LIN {X 0,Y 516.191,Z 499.318,A -85,B 0,C 180,E1 -4981.156,E2 -4981.156} C_VEL
LIN {X 0,Y 516.198,Z 499.528,A -85,B 0,C 180,E1 -4982.421,E2 -4982.421} C_VEL
LIN {X 0,Y 516.212,Z 498.459,A -85,B 0,C 180,E1 -4983.931,E2 -4983.931} C_VEL
LIN {X 0,Y 516.231,Z 496.319,A -85,B 0,C 180,E1 -4985.229,E2 -4985.229} C_VEL
LIN {X 0,Y 516.336,Z 492.856,A -85,B 0,C 180,E1 -4986.576,E2 -4986.576} C_VEL
LIN {X 0,Y 516.422,Z 488.222,A -85,B 0,C 180,E1 -4987.877,E2 -4987.877} C_VEL
LIN {X 0,Y 516.57,Z 482.317,A -85,B 0,C 180,E1 -4989.15,E2 -4989.15} C_VEL
LIN {X 0,Y 516.77,Z 474.967,A -85,B 0,C 180,E1 -4990.395,E2 -4990.395} C_VEL
LIN {X 0,Y 516.949,Z 467.344,A -85,B 0,C 180,E1 -4991.437,E2 -4991.437} C_VEL
LIN {X 0,Y 517.264,Z 457.539,A -85,B 0,C 180,E1 -4992.527,E2 -4992.527} C_VEL
LIN {X 0,Y 517.546,Z 447.499,A -85,B 0,C 180,E1 -4993.428,E2 -4993.428} C_VEL
LIN {X 0,Y 517.803,Z 437.525,A -85,B 0,C 180,E1 -4994.151,E2 -4994.151} C_VEL
LIN {X 0,Y 518.099,Z 426.299,A -85,B 0,C 180,E1 -4994.797,E2 -4994.797} C_VEL
LIN {X 0,Y 518.372,Z 414.041,A -85,B 0,C 180,E1 -4995.333,E2 -4995.333} C_VEL
LIN {X 0,Y 518.246,Z 407.392,A -85,B 0,C 180,E1 -4995.565,E2 -4995.565} C_VEL
LIN {X 0,Y 516.248,Z 397.17,A -85,B 0,C 180,E1 -4995.893,E2 -4995.893} C_VEL
LIN {X 0,Y 516.275,Z 394.338,A -85,B 0,C 180,E1 -4998.478,E2 -4998.478} C_VEL
LIN {X 0,Y 516.29,Z 391.343,A -85,B 0,C 180,E1 -5001.231,E2 -5001.231} C_VEL
LIN {X 0,Y 516.378,Z 388.125,A -85,B 0,C 180,E1 -5004.18,E2 -5004.18} C_VEL
LIN {X 0,Y 516.457,Z 385.062,A -85,B 0,C 180,E1 -5007.021,E2 -5007.021} C_VEL
LIN {X 0,Y 516.53,Z 382.092,A -85,B 0,C 180,E1 -5009.773,E2 -5009.773} C_VEL
LIN {X 0,Y 516.548,Z 379.223,A -85,B 0,C 180,E1 -5012.445,E2 -5012.445} C_VEL
LIN {X 0,Y 516.602,Z 376.37,A -85,B 0,C 180,E1 -5015.056,E2 -5015.056} C_VEL
LIN {X 0,Y 516.777,Z 376.119,A -85,B 0,C 180,E1 -5016.772,E2 -5016.772} C_VEL
LIN {X 0,Y 516.934,Z 376.098,A -85,B 0,C 180,E1 -5019.731,E2 -5019.731} C_VEL
LIN {X 0,Y 516.923,Z 376.096,A -85,B 0,C 180,E1 -5022.596,E2 -5022.596} C_VEL
LIN {X 0,Y 516.936,Z 376.095,A -85,B 0,C 180,E1 -5025.03,E2 -5025.03} C_VEL
LIN {X 0,Y 516.959,Z 376.094,A -85,B 0,C 180,E1 -5028.233,E2 -5028.233} C_VEL
LIN {X 0,Y 516.964,Z 376.091,A -85,B 0,C 180,E1 -5031.399,E2 -5031.399} C_VEL
LIN {X 0,Y 517.004,Z 376.086,A -85,B 0,C 180,E1 -5033.757,E2 -5033.757} C_VEL
LIN {X 0,Y 517.079,Z 376.076,A -85,B 0,C 180,E1 -5037.663,E2 -5037.663} C_VEL
LIN {X 0,Y 517.09,Z 376.075,A -85,B 0,C 180,E1 -5040.779,E2 -5040.779} C_VEL
LIN {X 0,Y 517.009,Z 376.086,A -85,B 0,C 180,E1 -5043.117,E2 -5043.117} C_VEL
LIN {X 0,Y 517.003,Z 376.087,A -85,B 0,C 180,E1 -5046.243,E2 -5046.243} C_VEL
LIN {X 0,Y 516.949,Z 376.092,A -85,B 0,C 180,E1 -5049.389,E2 -5049.389} C_VEL
LIN {X 0,Y 516.951,Z 376.092,A -85,B 0,C 180,E1 -5051.81,E2 -5051.81} C_VEL
LIN {X 0,Y 516.938,Z 376.094,A -85,B 0,C 180,E1 -5055.147,E2 -5055.147} C_VEL
LIN {X 0,Y 516.92,Z 376.097,A -85,B 0,C 180,E1 -5058.222,E2 -5058.222} C_VEL
LIN {X 0,Y 516.906,Z 376.099,A -85,B 0,C 180,E1 -5060.702,E2 -5060.702} C_VEL
LIN {X 0,Y 516.906,Z 376.098,A -85,B 0,C 180,E1 -5064.072,E2 -5064.072} C_VEL
LIN {X 0,Y 516.924,Z 376.095,A -85,B 0,C 180,E1 -5066.658,E2 -5066.658} C_VEL
LIN {X 0,Y 516.906,Z 376.101,A -85,B 0,C 180,E1 -5069.524,E2 -5069.524} C_VEL
LIN {X 0,Y 516.889,Z 376.101,A -85,B 0,C 180,E1 -5072.543,E2 -5072.543} C_VEL
LIN {X 0,Y 516.862,Z 376.106,A -85,B 0,C 180,E1 -5075.33,E2 -5075.33} C_VEL
LIN {X 0,Y 516.877,Z 376.105,A -85,B 0,C 180,E1 -5077.944,E2 -5077.944} C_VEL
LIN {X 0,Y 516.901,Z 376.1,A -85,B 0,C 180,E1 -5080.74,E2 -5080.74} C_VEL
LIN {X 0,Y 516.879,Z 376.105,A -85,B 0,C 180,E1 -5083.904,E2 -5083.904} C_VEL
LIN {X 0,Y 516.88,Z 376.104,A -85,B 0,C 180,E1 -5086.107,E2 -5086.107} C_VEL
LIN {X 0,Y 516.894,Z 376.102,A -85,B 0,C 180,E1 -5089.26,E2 -5089.26} C_VEL
LIN {X 0,Y 516.898,Z 376.203,A -85,B 0,C 180,E1 -5091.227,E2 -5091.227} C_VEL
LIN {X 0,Y 518.101,Z 382.793,A -85,B 0,C 180,E1 -5093.838,E2 -5093.838} C_VEL
LIN {X 0,Y 518.058,Z 388.209,A -85,B 0,C 180,E1 -5095.846,E2 -5095.846} C_VEL
LIN {X 0,Y 517.781,Z 396.952,A -85,B 0,C 180,E1 -5098.773,E2 -5098.773} C_VEL
LIN {X 0,Y 517.567,Z 406.705,A -85,B 0,C 180,E1 -5101.962,E2 -5101.962} C_VEL
LIN {X 0,Y 517.319,Z 414.959,A -85,B 0,C 180,E1 -5104.663,E2 -5104.663} C_VEL
LIN {X 0,Y 517.116,Z 424.226,A -85,B 0,C 180,E1 -5107.633,E2 -5107.633} C_VEL
LIN {X 0,Y 516.907,Z 433.493,A -85,B 0,C 180,E1 -5110.543,E2 -5110.543} C_VEL
LIN {X 0,Y 516.712,Z 442.76,A -85,B 0,C 180,E1 -5113.404,E2 -5113.404} C_VEL
LIN {X 0,Y 516.591,Z 451.736,A -85,B 0,C 180,E1 -5116.095,E2 -5116.095} C_VEL
LIN {X 0,Y 518.517,Z 464.185,A -85,B 0,C 180,E1 -5116.429,E2 -5116.429} C_VEL
LIN {X 0,Y 518.247,Z 476.985,A -85,B 0,C 180,E1 -5116.871,E2 -5116.871} C_VEL
LIN {X 0,Y 517.949,Z 489.176,A -85,B 0,C 180,E1 -5117.461,E2 -5117.461} C_VEL
LIN {X 0,Y 517.703,Z 500.576,A -85,B 0,C 180,E1 -5118.179,E2 -5118.179} C_VEL
LIN {X 0,Y 517.38,Z 511.401,A -85,B 0,C 180,E1 -5119.037,E2 -5119.037} C_VEL
LIN {X 0,Y 517.045,Z 521.335,A -85,B 0,C 180,E1 -5120.02,E2 -5120.02} C_VEL
LIN {X 0,Y 516.814,Z 530.96,A -85,B 0,C 180,E1 -5121.2,E2 -5121.2} C_VEL
LIN {X 0,Y 516.563,Z 538.621,A -85,B 0,C 180,E1 -5122.377,E2 -5122.377} C_VEL
LIN {X 0,Y 516.427,Z 545.679,A -85,B 0,C 180,E1 -5123.75,E2 -5123.75} C_VEL
LIN {X 0,Y 516.313,Z 550.372,A -85,B 0,C 180,E1 -5124.924,E2 -5124.924} C_VEL
LIN {X 0,Y 516.355,Z 553.957,A -85,B 0,C 180,E1 -5126.098,E2 -5126.098} C_VEL
LIN {X 0,Y 516.282,Z 555.807,A -85,B 0,C 180,E1 -5126.879,E2 -5126.879} C_VEL
LIN {X 0,Y 516.261,Z 557.196,A -85,B 0,C 180,E1 -5127.659,E2 -5127.659} C_VEL
LIN {X 0,Y 516.16,Z 558.785,A -85,B 0,C 180,E1 -5129.22,E2 -5129.22} C_VEL
LIN {X 0,Y 516.154,Z 559,A -85,B 0,C 180,E1 -5130,E2 -5130} C_VEL
LIN {X 0,Y 516.192,Z 558.186,A -85,B 0,C 180,E1 -5131.56,E2 -5131.56} C_VEL
LIN {X 0,Y 516.261,Z 557.199,A -85,B 0,C 180,E1 -5132.34,E2 -5132.34} C_VEL
LIN {X 0,Y 516.282,Z 555.81,A -85,B 0,C 180,E1 -5133.121,E2 -5133.121} C_VEL
LIN {X 0,Y 516.344,Z 552.896,A -85,B 0,C 180,E1 -5134.293,E2 -5134.293} C_VEL
LIN {X 0,Y 516.405,Z 548.95,A -85,B 0,C 180,E1 -5135.466,E2 -5135.466} C_VEL
LIN {X 0,Y 516.486,Z 543.035,A -85,B 0,C 180,E1 -5136.807,E2 -5136.807} C_VEL
LIN {X 0,Y 516.64,Z 536.239,A -85,B 0,C 180,E1 -5138.015,E2 -5138.015} C_VEL
LIN {X 0,Y 516.867,Z 527.994,A -85,B 0,C 180,E1 -5139.193,E2 -5139.193} C_VEL
LIN {X 0,Y 517.078,Z 519.543,A -85,B 0,C 180,E1 -5140.177,E2 -5140.177} C_VEL
LIN {X 0,Y 517.474,Z 509.101,A -85,B 0,C 180,E1 -5141.159,E2 -5141.159} C_VEL
LIN {X 0,Y 517.718,Z 497.634,A -85,B 0,C 180,E1 -5142.026,E2 -5142.026} C_VEL
LIN {X 0,Y 517.981,Z 487.416,A -85,B 0,C 180,E1 -5142.637,E2 -5142.637} C_VEL
LIN {X 0,Y 518.269,Z 475.776,A -85,B 0,C 180,E1 -5143.178,E2 -5143.178} C_VEL
LIN {X 0,Y 518.44,Z 462.821,A -85,B 0,C 180,E1 -5143.61,E2 -5143.61} C_VEL
LIN {X 0,Y 516.574,Z 451.532,A -85,B 0,C 180,E1 -5143.924,E2 -5143.924} C_VEL
LIN {X 0,Y 516.712,Z 442.761,A -85,B 0,C 180,E1 -5146.596,E2 -5146.596} C_VEL
LIN {X 0,Y 516.906,Z 433.494,A -85,B 0,C 180,E1 -5149.457,E2 -5149.457} C_VEL
LIN {X 0,Y 517.096,Z 423.966,A -85,B 0,C 180,E1 -5152.45,E2 -5152.45} C_VEL
LIN {X 0,Y 517.371,Z 413.636,A -85,B 0,C 180,E1 -5155.765,E2 -5155.765} C_VEL
LIN {X 0,Y 517.598,Z 404.312,A -85,B 0,C 180,E1 -5158.817,E2 -5158.817} C_VEL
LIN {X 0,Y 517.836,Z 396.125,A -85,B 0,C 180,E1 -5161.547,E2 -5161.547} C_VEL
LIN {X 0,Y 518.098,Z 388.482,A -85,B 0,C 180,E1 -5164.161,E2 -5164.161} C_VEL
LIN {X 0,Y 518.11,Z 382.817,A -85,B 0,C 180,E1 -5166.16,E2 -5166.16} C_VEL
LIN {X 0,Y 516.893,Z 376.1,A -85,B 0,C 180,E1 -5168.892,E2 -5168.892} C_VEL
LIN {X 0,Y 516.91,Z 376.099,A -85,B 0,C 180,E1 -5171.774,E2 -5171.774} C_VEL
LIN {X 0,Y 516.918,Z 376.099,A -85,B 0,C 180,E1 -5175.009,E2 -5175.009} C_VEL
LIN {X 0,Y 516.917,Z 376.099,A -85,B 0,C 180,E1 -5178.397,E2 -5178.397} C_VEL
LIN {X 0,Y 516.881,Z 376.102,A -85,B 0,C 180,E1 -5181.284,E2 -5181.284} C_VEL
LIN {X 0,Y 516.885,Z 376.102,A -85,B 0,C 180,E1 -5184.221,E2 -5184.221} C_VEL
LIN {X 0,Y 516.892,Z 376.102,A -85,B 0,C 180,E1 -5187.053,E2 -5187.053} C_VEL
LIN {X 0,Y 516.885,Z 376.1,A -85,B 0,C 180,E1 -5189.796,E2 -5189.796} C_VEL
LIN {X 0,Y 516.923,Z 376.096,A -85,B 0,C 180,E1 -5192.467,E2 -5192.467} C_VEL
LIN {X 0,Y 516.903,Z 376.101,A -85,B 0,C 180,E1 -5195.071,E2 -5195.071} C_VEL
LIN {X 0,Y 516.878,Z 376.104,A -85,B 0,C 180,E1 -5198.462,E2 -5198.462} C_VEL
LIN {X 0,Y 516.897,Z 376.1,A -85,B 0,C 180,E1 -5200.955,E2 -5200.955} C_VEL
LIN {X 0,Y 516.909,Z 376.098,A -85,B 0,C 180,E1 -5203.41,E2 -5203.41} C_VEL
LIN {X 0,Y 516.886,Z 376.101,A -85,B 0,C 180,E1 -5205.833,E2 -5205.833} C_VEL
LIN {X 0,Y 516.948,Z 376.094,A -85,B 0,C 180,E1 -5209.028,E2 -5209.028} C_VEL
LIN {X 0,Y 516.97,Z 376.09,A -85,B 0,C 180,E1 -5212.187,E2 -5212.187} C_VEL
LIN {X 0,Y 517.02,Z 376.085,A -85,B 0,C 180,E1 -5214.54,E2 -5214.54} C_VEL
LIN {X 0,Y 517.074,Z 376.076,A -85,B 0,C 180,E1 -5217.663,E2 -5217.663} C_VEL
LIN {X 0,Y 517.088,Z 376.076,A -85,B 0,C 180,E1 -5220.779,E2 -5220.779} C_VEL
LIN {X 0,Y 517.008,Z 376.085,A -85,B 0,C 180,E1 -5223.117,E2 -5223.117} C_VEL
LIN {X 0,Y 517.002,Z 376.088,A -85,B 0,C 180,E1 -5226.243,E2 -5226.243} C_VEL
LIN {X 0,Y 516.95,Z 376.093,A -85,B 0,C 180,E1 -5229.389,E2 -5229.389} C_VEL
LIN {X 0,Y 516.948,Z 376.094,A -85,B 0,C 180,E1 -5231.811,E2 -5231.811} C_VEL
LIN {X 0,Y 516.935,Z 376.094,A -85,B 0,C 180,E1 -5235.147,E2 -5235.147} C_VEL
LIN {X 0,Y 516.917,Z 376.099,A -85,B 0,C 180,E1 -5238.223,E2 -5238.223} C_VEL
LIN {X 0,Y 516.905,Z 376.099,A -85,B 0,C 180,E1 -5240.702,E2 -5240.702} C_VEL
LIN {X 0,Y 516.903,Z 376.1,A -85,B 0,C 180,E1 -5244.073,E2 -5244.073} C_VEL
LIN {X 0,Y 516.922,Z 376.097,A -85,B 0,C 180,E1 -5246.658,E2 -5246.658} C_VEL
LIN {X 0,Y 516.904,Z 376.099,A -85,B 0,C 180,E1 -5249.525,E2 -5249.525} C_VEL
LIN {X 0,Y 516.895,Z 376.102,A -85,B 0,C 180,E1 -5252.545,E2 -5252.545} C_VEL
LIN {X 0,Y 516.879,Z 376.1,A -85,B 0,C 180,E1 -5255.333,E2 -5255.333} C_VEL
LIN {X 0,Y 516.877,Z 376.103,A -85,B 0,C 180,E1 -5257.944,E2 -5257.944} C_VEL
LIN {X 0,Y 516.9,Z 376.099,A -85,B 0,C 180,E1 -5260.74,E2 -5260.74} C_VEL
LIN {X 0,Y 516.878,Z 376.103,A -85,B 0,C 180,E1 -5263.904,E2 -5263.904} C_VEL
LIN {X 0,Y 516.879,Z 376.103,A -85,B 0,C 180,E1 -5266.108,E2 -5266.108} C_VEL
LIN {X 0,Y 516.915,Z 376.098,A -85,B 0,C 180,E1 -5268.399,E2 -5268.399} C_VEL
LIN {X 0,Y 516.879,Z 376.104,A -85,B 0,C 180,E1 -5270.307,E2 -5270.307} C_VEL
LIN {X 0,Y 516.21,Z 376.185,A -85,B 0,C 180,E1 -5270.957,E2 -5270.957} C_VEL
LIN {X 0,Y 513.365,Z 376.54,A -85,B 0,C 180,E1 -5272.013,E2 -5272.013} C_VEL
LIN {X 0,Y 510.957,Z 376.842,A -85,B 0,C 180,E1 -5272.863,E2 -5272.863} C_VEL
LIN {X 0,Y 509.917,Z 376.971,A -85,B 0,C 180,E1 -5273.52,E2 -5273.52} C_VEL
LIN {X 0,Y 509.828,Z 376.981,A -85,B 0,C 180,E1 -5273.742,E2 -5273.742} C_VEL
LIN {X 0,Y 509.861,Z 376.977,A -85,B 0,C 180,E1 -5276.54,E2 -5276.54} C_VEL
LIN {X 0,Y 509.846,Z 376.979,A -85,B 0,C 180,E1 -5279.335,E2 -5279.335} C_VEL
LIN {X 0,Y 509.894,Z 376.973,A -85,B 0,C 180,E1 -5282.055,E2 -5282.055} C_VEL
LIN {X 0,Y 509.879,Z 376.974,A -85,B 0,C 180,E1 -5284.705,E2 -5284.705} C_VEL
LIN {X 0,Y 509.839,Z 376.979,A -85,B 0,C 180,E1 -5287.456,E2 -5287.456} C_VEL
LIN {X 0,Y 509.919,Z 376.969,A -85,B 0,C 180,E1 -5289.845,E2 -5289.845} C_VEL
LIN {X 0,Y 509.883,Z 376.972,A -85,B 0,C 180,E1 -5293.175,E2 -5293.175} C_VEL
LIN {X 0,Y 509.868,Z 376.976,A -85,B 0,C 180,E1 -5295.635,E2 -5295.635} C_VEL
LIN {X 0,Y 509.917,Z 376.969,A -85,B 0,C 180,E1 -5298.875,E2 -5298.875} C_VEL
LIN {X 0,Y 509.955,Z 376.965,A -85,B 0,C 180,E1 -5302.079,E2 -5302.079} C_VEL
LIN {X 0,Y 509.986,Z 376.961,A -85,B 0,C 180,E1 -5304.465,E2 -5304.465} C_VEL
LIN {X 0,Y 509.828,Z 376.984,A -85,B 0,C 180,E1 -5308.42,E2 -5308.42} C_VEL
LIN {X 0,Y 509.779,Z 376.991,A -85,B 0,C 180,E1 -5309.21,E2 -5309.21} C_VEL
LIN {X 0,Y 509.632,Z 378.352,A -85,B 0,C 180,E1 -5310.79,E2 -5310.79} C_VEL
LIN {X 0,Y 509.491,Z 382.661,A -85,B 0,C 180,E1 -5314.748,E2 -5314.748} C_VEL
LIN {X 0,Y 509.445,Z 385.291,A -85,B 0,C 180,E1 -5317.132,E2 -5317.132} C_VEL
LIN {X 0,Y 509.358,Z 388.826,A -85,B 0,C 180,E1 -5320.333,E2 -5320.333} C_VEL
LIN {X 0,Y 509.291,Z 391.515,A -85,B 0,C 180,E1 -5322.756,E2 -5322.756} C_VEL
LIN {X 0,Y 509.302,Z 394.318,A -85,B 0,C 180,E1 -5325.2,E2 -5325.2} C_VEL
LIN {X 0,Y 509.21,Z 397.43,A -85,B 0,C 180,E1 -5328.014,E2 -5328.014} C_VEL
LIN {X 0,Y 511.466,Z 408.493,A -85,B 0,C 180,E1 -5328.372,E2 -5328.372} C_VEL
LIN {X 0,Y 511.353,Z 420.799,A -85,B 0,C 180,E1 -5328.843,E2 -5328.843} C_VEL
LIN {X 0,Y 511.021,Z 433.18,A -85,B 0,C 180,E1 -5329.482,E2 -5329.482} C_VEL
LIN {X 0,Y 510.748,Z 444.58,A -85,B 0,C 180,E1 -5330.256,E2 -5330.256} C_VEL
LIN {X 0,Y 510.386,Z 455.513,A -85,B 0,C 180,E1 -5331.19,E2 -5331.19} C_VEL
LIN {X 0,Y 510.048,Z 465.493,A -85,B 0,C 180,E1 -5332.253,E2 -5332.253} C_VEL
LIN {X 0,Y 509.729,Z 473.801,A -85,B 0,C 180,E1 -5333.353,E2 -5333.353} C_VEL
LIN {X 0,Y 509.56,Z 481.606,A -85,B 0,C 180,E1 -5334.637,E2 -5334.637} C_VEL
LIN {X 0,Y 509.419,Z 487.051,A -85,B 0,C 180,E1 -5335.758,E2 -5335.758} C_VEL
LIN {X 0,Y 509.286,Z 492.135,A -85,B 0,C 180,E1 -5337.09,E2 -5337.09} C_VEL
LIN {X 0,Y 509.216,Z 495.877,A -85,B 0,C 180,E1 -5338.434,E2 -5338.434} C_VEL
LIN {X 0,Y 509.151,Z 498.412,A -85,B 0,C 180,E1 -5339.796,E2 -5339.796} C_VEL
LIN {X 0,Y 509.114,Z 499.749,A -85,B 0,C 180,E1 -5341.143,E2 -5341.143} C_VEL
LIN {X 0,Y 509.103,Z 499.922,A -85,B 0,C 180,E1 -5342.639,E2 -5342.639} C_VEL
LIN {X 0,Y 509.122,Z 498.729,A -85,B 0,C 180,E1 -5344.08,E2 -5344.08} C_VEL
LIN {X 0,Y 509.184,Z 496.303,A -85,B 0,C 180,E1 -5345.477,E2 -5345.477} C_VEL
LIN {X 0,Y 509.281,Z 492.696,A -85,B 0,C 180,E1 -5346.832,E2 -5346.832} C_VEL
LIN {X 0,Y 509.403,Z 487.894,A -85,B 0,C 180,E1 -5348.149,E2 -5348.149} C_VEL
LIN {X 0,Y 509.573,Z 481.777,A -85,B 0,C 180,E1 -5349.434,E2 -5349.434} C_VEL
LIN {X 0,Y 509.787,Z 474.19,A -85,B 0,C 180,E1 -5350.69,E2 -5350.69} C_VEL
LIN {X 0,Y 510.061,Z 465.702,A -85,B 0,C 180,E1 -5351.823,E2 -5351.823} C_VEL
LIN {X 0,Y 510.323,Z 456.477,A -85,B 0,C 180,E1 -5352.822,E2 -5352.822} C_VEL
LIN {X 0,Y 510.672,Z 445.775,A -85,B 0,C 180,E1 -5353.752,E2 -5353.752} C_VEL
LIN {X 0,Y 510.944,Z 434.354,A -85,B 0,C 180,E1 -5354.547,E2 -5354.547} C_VEL
LIN {X 0,Y 511.274,Z 422.583,A -85,B 0,C 180,E1 -5355.176,E2 -5355.176} C_VEL
LIN {X 0,Y 511.513,Z 409.334,A -85,B 0,C 180,E1 -5355.695,E2 -5355.695} C_VEL
LIN {X 0,Y 509.588,Z 399.448,A -85,B 0,C 180,E1 -5356.024,E2 -5356.024} C_VEL
LIN {X 0,Y 509.179,Z 397.637,A -85,B 0,C 180,E1 -5356.088,E2 -5356.088} C_VEL
LIN {X 0,Y 509.207,Z 394.981,A -85,B 0,C 180,E1 -5358.51,E2 -5358.51} C_VEL
LIN {X 0,Y 509.232,Z 391.61,A -85,B 0,C 180,E1 -5361.607,E2 -5361.607} C_VEL
LIN {X 0,Y 509.344,Z 388.36,A -85,B 0,C 180,E1 -5364.583,E2 -5364.583} C_VEL
LIN {X 0,Y 509.419,Z 385.318,A -85,B 0,C 180,E1 -5367.449,E2 -5367.449} C_VEL
LIN {X 0,Y 509.465,Z 382.195,A -85,B 0,C 180,E1 -5370.35,E2 -5370.35} C_VEL
LIN {X 0,Y 509.494,Z 379.428,A -85,B 0,C 180,E1 -5372.922,E2 -5372.922} C_VEL
LIN {X 0,Y 509.528,Z 377.548,A -85,B 0,C 180,E1 -5374.685,E2 -5374.685} C_VEL
LIN {X 0,Y 509.61,Z 377.01,A -85,B 0,C 180,E1 -5375.561,E2 -5375.561} C_VEL
LIN {X 0,Y 509.816,Z 376.984,A -85,B 0,C 180,E1 -5378.148,E2 -5378.148} C_VEL
LIN {X 0,Y 509.86,Z 376.978,A -85,B 0,C 180,E1 -5380.681,E2 -5380.681} C_VEL
LIN {X 0,Y 509.879,Z 376.975,A -85,B 0,C 180,E1 -5383.174,E2 -5383.174} C_VEL
LIN {X 0,Y 509.857,Z 376.978,A -85,B 0,C 180,E1 -5385.634,E2 -5385.634} C_VEL
LIN {X 0,Y 509.911,Z 376.969,A -85,B 0,C 180,E1 -5388.874,E2 -5388.874} C_VEL
LIN {X 0,Y 509.945,Z 376.965,A -85,B 0,C 180,E1 -5392.078,E2 -5392.078} C_VEL
LIN {X 0,Y 509.977,Z 376.961,A -85,B 0,C 180,E1 -5394.464,E2 -5394.464} C_VEL
LIN {X 0,Y 510.049,Z 376.952,A -85,B 0,C 180,E1 -5397.631,E2 -5397.631} C_VEL
LIN {X 0,Y 510.06,Z 376.951,A -85,B 0,C 180,E1 -5400.789,E2 -5400.789} C_VEL
LIN {X 0,Y 509.951,Z 376.964,A -85,B 0,C 180,E1 -5403.16,E2 -5403.16} C_VEL
LIN {X 0,Y 509.971,Z 376.964,A -85,B 0,C 180,E1 -5406.33,E2 -5406.33} C_VEL
LIN {X 0,Y 509.91,Z 376.971,A -85,B 0,C 180,E1 -5408.72,E2 -5408.72} C_VEL
LIN {X 0,Y 509.899,Z 376.971,A -85,B 0,C 180,E1 -5411.932,E2 -5411.932} C_VEL
LIN {X 0,Y 509.887,Z 376.972,A -85,B 0,C 180,E1 -5415.242,E2 -5415.242} C_VEL
LIN {X 0,Y 509.883,Z 376.972,A -85,B 0,C 180,E1 -5418.001,E2 -5418.001} C_VEL
LIN {X 0,Y 509.844,Z 376.98,A -85,B 0,C 180,E1 -5421.002,E2 -5421.002} C_VEL
LIN {X 0,Y 509.865,Z 376.977,A -85,B 0,C 180,E1 -5424.426,E2 -5424.426} C_VEL
LIN {X 0,Y 509.883,Z 376.975,A -85,B 0,C 180,E1 -5427.056,E2 -5427.056} C_VEL
LIN {X 0,Y 509.852,Z 376.978,A -85,B 0,C 180,E1 -5429.751,E2 -5429.751} C_VEL
LIN {X 0,Y 509.862,Z 376.978,A -85,B 0,C 180,E1 -5432.773,E2 -5432.773} C_VEL
LIN {X 0,Y 509.821,Z 376.985,A -85,B 0,C 180,E1 -5435.579,E2 -5435.579} C_VEL
LIN {X 0,Y 509.855,Z 376.977,A -85,B 0,C 180,E1 -5438.338,E2 -5438.338} C_VEL
LIN {X 0,Y 509.863,Z 376.978,A -85,B 0,C 180,E1 -5441.425,E2 -5441.425} C_VEL
LIN {X 0,Y 509.854,Z 376.977,A -85,B 0,C 180,E1 -5444.668,E2 -5444.668} C_VEL
LIN {X 0,Y 509.857,Z 376.979,A -85,B 0,C 180,E1 -5448.103,E2 -5448.103} C_VEL
LIN {X 0,Y 509.882,Z 377.132,A -85,B 0,C 180,E1 -5450.97,E2 -5450.97} C_VEL
LIN {X 0,Y 511.155,Z 384.063,A -85,B 0,C 180,E1 -5453.757,E2 -5453.757} C_VEL
LIN {X 0,Y 511.097,Z 389.175,A -85,B 0,C 180,E1 -5455.683,E2 -5455.683} C_VEL
LIN {X 0,Y 510.803,Z 397.429,A -85,B 0,C 180,E1 -5458.544,E2 -5458.544} C_VEL
LIN {X 0,Y 510.548,Z 407.134,A -85,B 0,C 180,E1 -5461.763,E2 -5461.763} C_VEL
LIN {X 0,Y 510.298,Z 416.282,A -85,B 0,C 180,E1 -5464.727,E2 -5464.727} C_VEL
LIN {X 0,Y 510.079,Z 425.674,A -85,B 0,C 180,E1 -5467.775,E2 -5467.775} C_VEL
LIN {X 0,Y 509.86,Z 434.817,A -85,B 0,C 180,E1 -5470.682,E2 -5470.682} C_VEL
LIN {X 0,Y 509.648,Z 445.408,A -85,B 0,C 180,E1 -5473.991,E2 -5473.991} C_VEL
LIN {X 0,Y 509.544,Z 451.736,A -85,B 0,C 180,E1 -5475.899,E2 -5475.899} C_VEL
LIN {X 0,Y 511.549,Z 464.185,A -85,B 0,C 180,E1 -5476.24,E2 -5476.24} C_VEL
LIN {X 0,Y 511.336,Z 476.985,A -85,B 0,C 180,E1 -5476.69,E2 -5476.69} C_VEL
LIN {X 0,Y 511.001,Z 489.175,A -85,B 0,C 180,E1 -5477.288,E2 -5477.288} C_VEL
LIN {X 0,Y 510.727,Z 499.95,A -85,B 0,C 180,E1 -5477.971,E2 -5477.971} C_VEL
LIN {X 0,Y 510.404,Z 511.4,A -85,B 0,C 180,E1 -5478.885,E2 -5478.885} C_VEL
LIN {X 0,Y 510.03,Z 521.334,A -85,B 0,C 180,E1 -5479.881,E2 -5479.881} C_VEL
LIN {X 0,Y 509.76,Z 530.96,A -85,B 0,C 180,E1 -5481.077,E2 -5481.077} C_VEL
LIN {X 0,Y 509.522,Z 538.621,A -85,B 0,C 180,E1 -5482.271,E2 -5482.271} C_VEL
LIN {X 0,Y 509.336,Z 545.679,A -85,B 0,C 180,E1 -5483.662,E2 -5483.662} C_VEL
LIN {X 0,Y 509.248,Z 550.372,A -85,B 0,C 180,E1 -5484.853,E2 -5484.853} C_VEL
LIN {X 0,Y 509.253,Z 553.958,A -85,B 0,C 180,E1 -5486.043,E2 -5486.043} C_VEL
LIN {X 0,Y 509.2,Z 555.807,A -85,B 0,C 180,E1 -5486.835,E2 -5486.835} C_VEL
LIN {X 0,Y 509.161,Z 557.196,A -85,B 0,C 180,E1 -5487.627,E2 -5487.627} C_VEL
LIN {X 0,Y 509.073,Z 558.785,A -85,B 0,C 180,E1 -5489.209,E2 -5489.209} C_VEL
LIN {X 0,Y 509.065,Z 559,A -85,B 0,C 180,E1 -5490,E2 -5490} C_VEL
LIN {X 0,Y 509.112,Z 558.185,A -85,B 0,C 180,E1 -5491.582,E2 -5491.582} C_VEL
LIN {X 0,Y 509.161,Z 557.198,A -85,B 0,C 180,E1 -5492.373,E2 -5492.373} C_VEL
LIN {X 0,Y 509.2,Z 555.81,A -85,B 0,C 180,E1 -5493.165,E2 -5493.165} C_VEL
LIN {X 0,Y 509.234,Z 552.896,A -85,B 0,C 180,E1 -5494.353,E2 -5494.353} C_VEL
LIN {X 0,Y 509.344,Z 548.95,A -85,B 0,C 180,E1 -5495.542,E2 -5495.542} C_VEL
LIN {X 0,Y 509.41,Z 543.283,A -85,B 0,C 180,E1 -5496.853,E2 -5496.853} C_VEL
LIN {X 0,Y 509.584,Z 536.239,A -85,B 0,C 180,E1 -5498.126,E2 -5498.126} C_VEL
LIN {X 0,Y 509.846,Z 527.994,A -85,B 0,C 180,E1 -5499.321,E2 -5499.321} C_VEL
LIN {X 0,Y 510.069,Z 519.543,A -85,B 0,C 180,E1 -5500.318,E2 -5500.318} C_VEL
LIN {X 0,Y 510.501,Z 509.1,A -85,B 0,C 180,E1 -5501.313,E2 -5501.313} C_VEL
LIN {X 0,Y 510.747,Z 498.398,A -85,B 0,C 180,E1 -5502.138,E2 -5502.138} C_VEL
LIN {X 0,Y 511.04,Z 487.416,A -85,B 0,C 180,E1 -5502.812,E2 -5502.812} C_VEL
LIN {X 0,Y 511.348,Z 475.776,A -85,B 0,C 180,E1 -5503.36,E2 -5503.36} C_VEL
LIN {X 0,Y 511.459,Z 463.278,A -85,B 0,C 180,E1 -5503.787,E2 -5503.787} C_VEL
LIN {X 0,Y 509.533,Z 451.532,A -85,B 0,C 180,E1 -5504.12,E2 -5504.12} C_VEL
LIN {X 0,Y 509.716,Z 441.437,A -85,B 0,C 180,E1 -5507.244,E2 -5507.244} C_VEL
LIN {X 0,Y 509.922,Z 432.17,A -85,B 0,C 180,E1 -5510.154,E2 -5510.154} C_VEL
LIN {X 0,Y 510.111,Z 422.903,A -85,B 0,C 180,E1 -5513.119,E2 -5513.119} C_VEL
LIN {X 0,Y 510.367,Z 413.582,A -85,B 0,C 180,E1 -5516.145,E2 -5516.145} C_VEL
LIN {X 0,Y 510.614,Z 404.241,A -85,B 0,C 180,E1 -5519.249,E2 -5519.249} C_VEL
LIN {X 0,Y 510.915,Z 396.19,A -85,B 0,C 180,E1 -5521.977,E2 -5521.977} C_VEL
LIN {X 0,Y 511.185,Z 388.108,A -85,B 0,C 180,E1 -5524.795,E2 -5524.795} C_VEL
LIN {X 0,Y 511.159,Z 384.088,A -85,B 0,C 180,E1 -5526.242,E2 -5526.242} C_VEL
LIN {X 0,Y 509.857,Z 376.976,A -85,B 0,C 180,E1 -5529.159,E2 -5529.159} C_VEL
LIN {X 0,Y 509.854,Z 376.979,A -85,B 0,C 180,E1 -5531.896,E2 -5531.896} C_VEL
LIN {X 0,Y 509.852,Z 376.979,A -85,B 0,C 180,E1 -5535.331,E2 -5535.331} C_VEL
LIN {X 0,Y 509.86,Z 376.978,A -85,B 0,C 180,E1 -5538.575,E2 -5538.575} C_VEL
LIN {X 0,Y 509.846,Z 376.98,A -85,B 0,C 180,E1 -5541.661,E2 -5541.661} C_VEL
LIN {X 0,Y 509.84,Z 376.979,A -85,B 0,C 180,E1 -5544.623,E2 -5544.623} C_VEL
LIN {X 0,Y 509.859,Z 376.976,A -85,B 0,C 180,E1 -5547.481,E2 -5547.481} C_VEL
LIN {X 0,Y 509.851,Z 376.977,A -85,B 0,C 180,E1 -5550.273,E2 -5550.273} C_VEL
LIN {X 0,Y 509.88,Z 376.975,A -85,B 0,C 180,E1 -5552.944,E2 -5552.944} C_VEL
LIN {X 0,Y 509.862,Z 376.975,A -85,B 0,C 180,E1 -5555.574,E2 -5555.574} C_VEL
LIN {X 0,Y 509.814,Z 376.981,A -85,B 0,C 180,E1 -5558.148,E2 -5558.148} C_VEL
LIN {X 0,Y 509.857,Z 376.979,A -85,B 0,C 180,E1 -5560.681,E2 -5560.681} C_VEL
LIN {X 0,Y 509.878,Z 376.974,A -85,B 0,C 180,E1 -5563.175,E2 -5563.175} C_VEL
LIN {X 0,Y 509.854,Z 376.976,A -85,B 0,C 180,E1 -5565.634,E2 -5565.634} C_VEL
LIN {X 0,Y 509.909,Z 376.97,A -85,B 0,C 180,E1 -5568.874,E2 -5568.874} C_VEL
LIN {X 0,Y 509.943,Z 376.966,A -85,B 0,C 180,E1 -5572.078,E2 -5572.078} C_VEL
LIN {X 0,Y 509.972,Z 376.962,A -85,B 0,C 180,E1 -5574.464,E2 -5574.464} C_VEL
LIN {X 0,Y 510.046,Z 376.952,A -85,B 0,C 180,E1 -5577.631,E2 -5577.631} C_VEL
LIN {X 0,Y 510.058,Z 376.952,A -85,B 0,C 180,E1 -5580.79,E2 -5580.79} C_VEL
LIN {X 0,Y 509.95,Z 376.964,A -85,B 0,C 180,E1 -5583.16,E2 -5583.16} C_VEL
LIN {X 0,Y 509.97,Z 376.963,A -85,B 0,C 180,E1 -5586.33,E2 -5586.33} C_VEL
LIN {X 0,Y 509.91,Z 376.97,A -85,B 0,C 180,E1 -5588.72,E2 -5588.72} C_VEL
LIN {X 0,Y 509.896,Z 376.972,A -85,B 0,C 180,E1 -5591.932,E2 -5591.932} C_VEL
LIN {X 0,Y 509.884,Z 376.972,A -85,B 0,C 180,E1 -5595.242,E2 -5595.242} C_VEL
LIN {X 0,Y 509.88,Z 376.974,A -85,B 0,C 180,E1 -5598.002,E2 -5598.002} C_VEL
LIN {X 0,Y 509.843,Z 376.978,A -85,B 0,C 180,E1 -5601.002,E2 -5601.002} C_VEL
LIN {X 0,Y 509.829,Z 376.98,A -85,B 0,C 180,E1 -5603.564,E2 -5603.564} C_VEL
LIN {X 0,Y 509.906,Z 376.971,A -85,B 0,C 180,E1 -5606.38,E2 -5606.38} C_VEL
LIN {X 0,Y 509.87,Z 376.975,A -85,B 0,C 180,E1 -5608.845,E2 -5608.845} C_VEL
LIN {X 0,Y 509.819,Z 376.982,A -85,B 0,C 180,E1 -5611.59,E2 -5611.59} C_VEL
LIN {X 0,Y 509.849,Z 376.978,A -85,B 0,C 180,E1 -5614.414,E2 -5614.414} C_VEL
LIN {X 0,Y 509.815,Z 376.982,A -85,B 0,C 180,E1 -5617.341,E2 -5617.341} C_VEL
LIN {X 0,Y 509.857,Z 376.978,A -85,B 0,C 180,E1 -5620.381,E2 -5620.381} C_VEL
LIN {X 0,Y 509.818,Z 376.98,A -85,B 0,C 180,E1 -5623.063,E2 -5623.063} C_VEL
LIN {X 0,Y 509.827,Z 376.981,A -85,B 0,C 180,E1 -5625.793,E2 -5625.793} C_VEL
LIN {X 0,Y 509.856,Z 376.977,A -85,B 0,C 180,E1 -5628.576,E2 -5628.576} C_VEL
LIN {X 0,Y 509.849,Z 376.978,A -85,B 0,C 180,E1 -5631.787,E2 -5631.787} C_VEL
LIN {X 0,Y 509.828,Z 376.981,A -85,B 0,C 180,E1 -5633.742,E2 -5633.742} C_VEL
LIN {X 0,Y 509.162,Z 377.064,A -85,B 0,C 180,E1 -5634.402,E2 -5634.402} C_VEL
LIN {X 0,Y 506.346,Z 377.413,A -85,B 0,C 180,E1 -5635.474,E2 -5635.474} C_VEL
LIN {X 0,Y 503.954,Z 377.712,A -85,B 0,C 180,E1 -5636.337,E2 -5636.337} C_VEL
LIN {X 0,Y 502.905,Z 377.842,A -85,B 0,C 180,E1 -5637.004,E2 -5637.004} C_VEL
LIN {X 0,Y 502.808,Z 377.853,A -85,B 0,C 180,E1 -5637.229,E2 -5637.229} C_VEL
LIN {X 0,Y 502.815,Z 377.855,A -85,B 0,C 180,E1 -5640.066,E2 -5640.066} C_VEL
LIN {X 0,Y 502.834,Z 377.851,A -85,B 0,C 180,E1 -5642.534,E2 -5642.534} C_VEL
LIN {X 0,Y 502.831,Z 377.851,A -85,B 0,C 180,E1 -5645.299,E2 -5645.299} C_VEL
LIN {X 0,Y 502.787,Z 377.858,A -85,B 0,C 180,E1 -5647.827,E2 -5647.827} C_VEL
LIN {X 0,Y 502.826,Z 377.852,A -85,B 0,C 180,E1 -5650.401,E2 -5650.401} C_VEL
LIN {X 0,Y 502.831,Z 377.85,A -85,B 0,C 180,E1 -5652.932,E2 -5652.932} C_VEL
LIN {X 0,Y 502.849,Z 377.849,A -85,B 0,C 180,E1 -5655.43,E2 -5655.43} C_VEL
LIN {X 0,Y 502.881,Z 377.845,A -85,B 0,C 180,E1 -5658.717,E2 -5658.717} C_VEL
LIN {X 0,Y 502.905,Z 377.843,A -85,B 0,C 180,E1 -5661.967,E2 -5661.967} C_VEL
LIN {X 0,Y 502.942,Z 377.839,A -85,B 0,C 180,E1 -5664.387,E2 -5664.387} C_VEL
LIN {X 0,Y 502.802,Z 377.859,A -85,B 0,C 180,E1 -5668.398,E2 -5668.398} C_VEL
LIN {X 0,Y 502.628,Z 378.186,A -85,B 0,C 180,E1 -5670,E2 -5670} C_VEL
LIN {X 0,Y 502.474,Z 382.539,A -85,B 0,C 180,E1 -5674.01,E2 -5674.01} C_VEL
LIN {X 0,Y 502.443,Z 385.486,A -85,B 0,C 180,E1 -5676.72,E2 -5676.72} C_VEL
LIN {X 0,Y 502.271,Z 388.749,A -85,B 0,C 180,E1 -5679.666,E2 -5679.666} C_VEL
LIN {X 0,Y 502.258,Z 391.422,A -85,B 0,C 180,E1 -5682.116,E2 -5682.116} C_VEL
LIN {X 0,Y 502.205,Z 395.155,A -85,B 0,C 180,E1 -5685.42,E2 -5685.42} C_VEL
LIN {X 0,Y 502.156,Z 397.91,A -85,B 0,C 180,E1 -5687.815,E2 -5687.815} C_VEL
LIN {X 0,Y 504.627,Z 409.645,A -85,B 0,C 180,E1 -5688.21,E2 -5688.21} C_VEL
LIN {X 0,Y 504.424,Z 423.021,A -85,B 0,C 180,E1 -5688.743,E2 -5688.743} C_VEL
LIN {X 0,Y 504.087,Z 434.065,A -85,B 0,C 180,E1 -5689.337,E2 -5689.337} C_VEL
LIN {X 0,Y 503.813,Z 444.958,A -85,B 0,C 180,E1 -5690.091,E2 -5690.091} C_VEL
LIN {X 0,Y 503.441,Z 454.771,A -85,B 0,C 180,E1 -5690.929,E2 -5690.929} C_VEL
LIN {X 0,Y 503.128,Z 464.404,A -85,B 0,C 180,E1 -5691.941,E2 -5691.941} C_VEL
LIN {X 0,Y 502.796,Z 472.929,A -85,B 0,C 180,E1 -5693.04,E2 -5693.04} C_VEL
LIN {X 0,Y 502.582,Z 480.578,A -85,B 0,C 180,E1 -5694.27,E2 -5694.27} C_VEL
LIN {X 0,Y 502.358,Z 487.613,A -85,B 0,C 180,E1 -5695.702,E2 -5695.702} C_VEL
LIN {X 0,Y 502.237,Z 492.65,A -85,B 0,C 180,E1 -5697.051,E2 -5697.051} C_VEL
LIN {X 0,Y 502.146,Z 496.372,A -85,B 0,C 180,E1 -5698.415,E2 -5698.415} C_VEL
LIN {X 0,Y 502.068,Z 498.871,A -85,B 0,C 180,E1 -5699.786,E2 -5699.786} C_VEL
LIN {X 0,Y 502.048,Z 500.316,A -85,B 0,C 180,E1 -5701.359,E2 -5701.359} C_VEL
LIN {X 0,Y 502.023,Z 500.247,A -85,B 0,C 180,E1 -5702.863,E2 -5702.863} C_VEL
LIN {X 0,Y 502.05,Z 498.876,A -85,B 0,C 180,E1 -5704.318,E2 -5704.318} C_VEL
LIN {X 0,Y 502.15,Z 496.287,A -85,B 0,C 180,E1 -5705.732,E2 -5705.732} C_VEL
LIN {X 0,Y 502.226,Z 492.541,A -85,B 0,C 180,E1 -5707.094,E2 -5707.094} C_VEL
LIN {X 0,Y 502.386,Z 487.515,A -85,B 0,C 180,E1 -5708.427,E2 -5708.427} C_VEL
LIN {X 0,Y 502.55,Z 481.214,A -85,B 0,C 180,E1 -5709.721,E2 -5709.721} C_VEL
LIN {X 0,Y 502.808,Z 473.424,A -85,B 0,C 180,E1 -5710.993,E2 -5710.993} C_VEL
LIN {X 0,Y 503.114,Z 464.912,A -85,B 0,C 180,E1 -5712.106,E2 -5712.106} C_VEL
LIN {X 0,Y 503.422,Z 454.928,A -85,B 0,C 180,E1 -5713.161,E2 -5713.161} C_VEL
LIN {X 0,Y 503.727,Z 444.953,A -85,B 0,C 180,E1 -5714.016,E2 -5714.016} C_VEL
LIN {X 0,Y 504.06,Z 434.314,A -85,B 0,C 180,E1 -5714.75,E2 -5714.75} C_VEL
LIN {X 0,Y 504.427,Z 421.431,A -85,B 0,C 180,E1 -5715.429,E2 -5715.429} C_VEL
LIN {X 0,Y 504.538,Z 409.672,A -85,B 0,C 180,E1 -5715.889,E2 -5715.889} C_VEL
LIN {X 0,Y 502.802,Z 401.205,A -85,B 0,C 180,E1 -5716.185,E2 -5716.185} C_VEL
LIN {X 0,Y 502.107,Z 398.093,A -85,B 0,C 180,E1 -5716.282,E2 -5716.282} C_VEL
LIN {X 0,Y 502.147,Z 395.017,A -85,B 0,C 180,E1 -5719.092,E2 -5719.092} C_VEL
LIN {X 0,Y 502.171,Z 391.883,A -85,B 0,C 180,E1 -5721.99,E2 -5721.99} C_VEL
LIN {X 0,Y 502.286,Z 388.664,A -85,B 0,C 180,E1 -5724.993,E2 -5724.993} C_VEL
LIN {X 0,Y 502.379,Z 385.561,A -85,B 0,C 180,E1 -5727.886,E2 -5727.886} C_VEL
LIN {X 0,Y 502.4,Z 382.606,A -85,B 0,C 180,E1 -5730.685,E2 -5730.685} C_VEL
LIN {X 0,Y 502.445,Z 379.572,A -85,B 0,C 180,E1 -5733.533,E2 -5733.533} C_VEL
LIN {X 0,Y 502.551,Z 377.889,A -85,B 0,C 180,E1 -5735.366,E2 -5735.366} C_VEL
LIN {X 0,Y 502.76,Z 377.863,A -85,B 0,C 180,E1 -5737.825,E2 -5737.825} C_VEL
LIN {X 0,Y 502.821,Z 377.853,A -85,B 0,C 180,E1 -5740.4,E2 -5740.4} C_VEL
LIN {X 0,Y 502.828,Z 377.851,A -85,B 0,C 180,E1 -5742.931,E2 -5742.931} C_VEL
LIN {X 0,Y 502.839,Z 377.851,A -85,B 0,C 180,E1 -5745.429,E2 -5745.429} C_VEL
LIN {X 0,Y 502.875,Z 377.845,A -85,B 0,C 180,E1 -5748.717,E2 -5748.717} C_VEL
LIN {X 0,Y 502.896,Z 377.844,A -85,B 0,C 180,E1 -5751.966,E2 -5751.966} C_VEL
LIN {X 0,Y 502.933,Z 377.839,A -85,B 0,C 180,E1 -5754.386,E2 -5754.386} C_VEL
LIN {X 0,Y 503.019,Z 377.827,A -85,B 0,C 180,E1 -5757.598,E2 -5757.598} C_VEL
LIN {X 0,Y 503.03,Z 377.827,A -85,B 0,C 180,E1 -5760.8,E2 -5760.8} C_VEL
LIN {X 0,Y 502.894,Z 377.843,A -85,B 0,C 180,E1 -5763.204,E2 -5763.204} C_VEL
LIN {X 0,Y 502.921,Z 377.843,A -85,B 0,C 180,E1 -5766.419,E2 -5766.419} C_VEL
LIN {X 0,Y 502.869,Z 377.849,A -85,B 0,C 180,E1 -5768.843,E2 -5768.843} C_VEL
LIN {X 0,Y 502.84,Z 377.85,A -85,B 0,C 180,E1 -5772.102,E2 -5772.102} C_VEL
LIN {X 0,Y 502.842,Z 377.849,A -85,B 0,C 180,E1 -5775.4,E2 -5775.4} C_VEL
LIN {X 0,Y 502.84,Z 377.85,A -85,B 0,C 180,E1 -5778.123,E2 -5778.123} C_VEL
LIN {X 0,Y 502.823,Z 377.852,A -85,B 0,C 180,E1 -5780.536,E2 -5780.536} C_VEL
LIN {X 0,Y 502.789,Z 377.857,A -85,B 0,C 180,E1 -5783.041,E2 -5783.041} C_VEL
LIN {X 0,Y 502.837,Z 377.853,A -85,B 0,C 180,E1 -5785.676,E2 -5785.676} C_VEL
LIN {X 0,Y 502.836,Z 377.851,A -85,B 0,C 180,E1 -5788.373,E2 -5788.373} C_VEL
LIN {X 0,Y 502.788,Z 377.857,A -85,B 0,C 180,E1 -5791.499,E2 -5791.499} C_VEL
LIN {X 0,Y 502.785,Z 377.86,A -85,B 0,C 180,E1 -5793.995,E2 -5793.995} C_VEL
LIN {X 0,Y 502.774,Z 377.86,A -85,B 0,C 180,E1 -5797.178,E2 -5797.178} C_VEL
LIN {X 0,Y 502.823,Z 377.855,A -85,B 0,C 180,E1 -5800.012,E2 -5800.012} C_VEL
LIN {X 0,Y 502.769,Z 377.859,A -85,B 0,C 180,E1 -5803.232,E2 -5803.232} C_VEL
LIN {X 0,Y 502.787,Z 377.858,A -85,B 0,C 180,E1 -5805.662,E2 -5805.662} C_VEL
LIN {X 0,Y 502.822,Z 377.856,A -85,B 0,C 180,E1 -5809.005,E2 -5809.005} C_VEL
LIN {X 0,Y 502.827,Z 377.878,A -85,B 0,C 180,E1 -5810.64,E2 -5810.64} C_VEL
LIN {X 0,Y 504.156,Z 385.026,A -85,B 0,C 180,E1 -5813.602,E2 -5813.602} C_VEL
LIN {X 0,Y 504.122,Z 390.69,A -85,B 0,C 180,E1 -5815.715,E2 -5815.715} C_VEL
LIN {X 0,Y 503.847,Z 397.897,A -85,B 0,C 180,E1 -5818.307,E2 -5818.307} C_VEL
LIN {X 0,Y 503.527,Z 407.894,A -85,B 0,C 180,E1 -5821.67,E2 -5821.67} C_VEL
LIN {X 0,Y 503.308,Z 416.01,A -85,B 0,C 180,E1 -5824.35,E2 -5824.35} C_VEL
LIN {X 0,Y 503.064,Z 425.002,A -85,B 0,C 180,E1 -5827.228,E2 -5827.228} C_VEL
LIN {X 0,Y 502.874,Z 433.493,A -85,B 0,C 180,E1 -5829.977,E2 -5829.977} C_VEL
LIN {X 0,Y 502.627,Z 442.76,A -85,B 0,C 180,E1 -5832.925,E2 -5832.925} C_VEL
LIN {X 0,Y 502.489,Z 451.582,A -85,B 0,C 180,E1 -5835.693,E2 -5835.693} C_VEL
LIN {X 0,Y 504.672,Z 465.098,A -85,B 0,C 180,E1 -5836.075,E2 -5836.075} C_VEL
LIN {X 0,Y 504.396,Z 478.113,A -85,B 0,C 180,E1 -5836.555,E2 -5836.555} C_VEL
LIN {X 0,Y 504.032,Z 490.559,A -85,B 0,C 180,E1 -5837.189,E2 -5837.189} C_VEL
LIN {X 0,Y 503.743,Z 501.589,A -85,B 0,C 180,E1 -5837.92,E2 -5837.92} C_VEL
LIN {X 0,Y 503.385,Z 512.469,A -85,B 0,C 180,E1 -5838.83,E2 -5838.83} C_VEL
LIN {X 0,Y 503.024,Z 521.334,A -85,B 0,C 180,E1 -5839.739,E2 -5839.739} C_VEL
LIN {X 0,Y 502.704,Z 530.96,A -85,B 0,C 180,E1 -5840.951,E2 -5840.951} C_VEL
LIN {X 0,Y 502.47,Z 538.621,A -85,B 0,C 180,E1 -5842.162,E2 -5842.162} C_VEL
LIN {X 0,Y 502.275,Z 545.679,A -85,B 0,C 180,E1 -5843.573,E2 -5843.573} C_VEL
LIN {X 0,Y 502.185,Z 550.372,A -85,B 0,C 180,E1 -5844.781,E2 -5844.781} C_VEL
LIN {X 0,Y 502.152,Z 553.958,A -85,B 0,C 180,E1 -5845.987,E2 -5845.987} C_VEL
LIN {X 0,Y 502.121,Z 555.807,A -85,B 0,C 180,E1 -5846.79,E2 -5846.79} C_VEL
LIN {X 0,Y 502.066,Z 557.195,A -85,B 0,C 180,E1 -5847.593,E2 -5847.593} C_VEL
LIN {X 0,Y 501.99,Z 558.786,A -85,B 0,C 180,E1 -5849.198,E2 -5849.198} C_VEL
LIN {X 0,Y 501.98,Z 559,A -85,B 0,C 180,E1 -5850,E2 -5850} C_VEL
LIN {X 0,Y 502.035,Z 558.185,A -85,B 0,C 180,E1 -5851.604,E2 -5851.604} C_VEL
LIN {X 0,Y 502.066,Z 557.198,A -85,B 0,C 180,E1 -5852.407,E2 -5852.407} C_VEL
LIN {X 0,Y 502.121,Z 555.81,A -85,B 0,C 180,E1 -5853.209,E2 -5853.209} C_VEL
LIN {X 0,Y 502.128,Z 552.896,A -85,B 0,C 180,E1 -5854.415,E2 -5854.415} C_VEL
LIN {X 0,Y 502.259,Z 548.95,A -85,B 0,C 180,E1 -5855.621,E2 -5855.621} C_VEL
LIN {X 0,Y 502.335,Z 542.978,A -85,B 0,C 180,E1 -5857.011,E2 -5857.011} C_VEL
LIN {X 0,Y 502.542,Z 536.238,A -85,B 0,C 180,E1 -5858.241,E2 -5858.241} C_VEL
LIN {X 0,Y 502.811,Z 527.994,A -85,B 0,C 180,E1 -5859.452,E2 -5859.452} C_VEL
LIN {X 0,Y 503.07,Z 519.543,A -85,B 0,C 180,E1 -5860.463,E2 -5860.463} C_VEL
LIN {X 0,Y 503.532,Z 509.099,A -85,B 0,C 180,E1 -5861.472,E2 -5861.472} C_VEL
LIN {X 0,Y 503.813,Z 497.275,A -85,B 0,C 180,E1 -5862.388,E2 -5862.388} C_VEL
LIN {X 0,Y 504.163,Z 485.499,A -85,B 0,C 180,E1 -5863.092,E2 -5863.092} C_VEL
LIN {X 0,Y 504.542,Z 473.179,A -85,B 0,C 180,E1 -5863.646,E2 -5863.646} C_VEL
LIN {X 0,Y 504.573,Z 464.192,A -85,B 0,C 180,E1 -5863.953,E2 -5863.953} C_VEL
LIN {X 0,Y 502.487,Z 451.532,A -85,B 0,C 180,E1 -5864.322,E2 -5864.322} C_VEL
LIN {X 0,Y 502.662,Z 441.437,A -85,B 0,C 180,E1 -5867.493,E2 -5867.493} C_VEL
LIN {X 0,Y 502.904,Z 431.83,A -85,B 0,C 180,E1 -5870.558,E2 -5870.558} C_VEL
LIN {X 0,Y 503.126,Z 422.903,A -85,B 0,C 180,E1 -5873.459,E2 -5873.459} C_VEL
LIN {X 0,Y 503.399,Z 413.349,A -85,B 0,C 180,E1 -5876.535,E2 -5876.535} C_VEL
LIN {X 0,Y 503.651,Z 404.164,A -85,B 0,C 180,E1 -5879.674,E2 -5879.674} C_VEL
LIN {X 0,Y 504.023,Z 394.774,A -85,B 0,C 180,E1 -5882.942,E2 -5882.942} C_VEL
LIN {X 0,Y 504.288,Z 386.705,A -85,B 0,C 180,E1 -5885.825,E2 -5885.825} C_VEL
LIN {X 0,Y 503.478,Z 381.505,A -85,B 0,C 180,E1 -5887.892,E2 -5887.892} C_VEL
LIN {X 0,Y 502.801,Z 377.856,A -85,B 0,C 180,E1 -5889.427,E2 -5889.427} C_VEL
LIN {X 0,Y 502.798,Z 377.857,A -85,B 0,C 180,E1 -5892.198,E2 -5892.198} C_VEL
LIN {X 0,Y 502.796,Z 377.857,A -85,B 0,C 180,E1 -5895.467,E2 -5895.467} C_VEL
LIN {X 0,Y 502.821,Z 377.853,A -85,B 0,C 180,E1 -5899.003,E2 -5899.003} C_VEL
LIN {X 0,Y 502.789,Z 377.857,A -85,B 0,C 180,E1 -5902.046,E2 -5902.046} C_VEL
LIN {X 0,Y 502.804,Z 377.858,A -85,B 0,C 180,E1 -5905.034,E2 -5905.034} C_VEL
LIN {X 0,Y 502.781,Z 377.856,A -85,B 0,C 180,E1 -5907.915,E2 -5907.915} C_VEL
LIN {X 0,Y 502.817,Z 377.856,A -85,B 0,C 180,E1 -5910.712,E2 -5910.712} C_VEL
LIN {X 0,Y 502.873,Z 377.846,A -85,B 0,C 180,E1 -5913.434,E2 -5913.434} C_VEL
LIN {X 0,Y 502.783,Z 377.858,A -85,B 0,C 180,E1 -5916.086,E2 -5916.086} C_VEL
LIN {X 0,Y 502.775,Z 377.86,A -85,B 0,C 180,E1 -5918.688,E2 -5918.688} C_VEL
LIN {X 0,Y 502.822,Z 377.853,A -85,B 0,C 180,E1 -5921.248,E2 -5921.248} C_VEL
LIN {X 0,Y 502.815,Z 377.854,A -85,B 0,C 180,E1 -5923.767,E2 -5923.767} C_VEL
LIN {X 0,Y 502.822,Z 377.854,A -85,B 0,C 180,E1 -5926.254,E2 -5926.254} C_VEL
LIN {X 0,Y 502.872,Z 377.847,A -85,B 0,C 180,E1 -5928.717,E2 -5928.717} C_VEL
LIN {X 0,Y 502.893,Z 377.844,A -85,B 0,C 180,E1 -5931.967,E2 -5931.967} C_VEL
LIN {X 0,Y 502.928,Z 377.84,A -85,B 0,C 180,E1 -5934.386,E2 -5934.386} C_VEL
LIN {X 0,Y 503.015,Z 377.827,A -85,B 0,C 180,E1 -5937.598,E2 -5937.598} C_VEL
LIN {X 0,Y 503.016,Z 377.828,A -85,B 0,C 180,E1 -5940,E2 -5940} C_VEL
LIN {X 0,Y 503.016,Z 377.829,A -85,B 0,C 180,E1 -5942.402,E2 -5942.402} C_VEL
LIN {X 0,Y 502.929,Z 377.838,A -85,B 0,C 180,E1 -5945.614,E2 -5945.614} C_VEL
LIN {X 0,Y 502.893,Z 377.844,A -85,B 0,C 180,E1 -5948.034,E2 -5948.034} C_VEL
LIN {X 0,Y 502.873,Z 377.847,A -85,B 0,C 180,E1 -5951.283,E2 -5951.283} C_VEL
LIN {X 0,Y 502.836,Z 377.852,A -85,B 0,C 180,E1 -5954.571,E2 -5954.571} C_VEL
LIN {X 0,Y 502.853,Z 377.848,A -85,B 0,C 180,E1 -5957.907,E2 -5957.907} C_VEL
LIN {X 0,Y 502.82,Z 377.854,A -85,B 0,C 180,E1 -5960.537,E2 -5960.537} C_VEL
LIN {X 0,Y 502.789,Z 377.856,A -85,B 0,C 180,E1 -5963.041,E2 -5963.041} C_VEL
LIN {X 0,Y 502.834,Z 377.85,A -85,B 0,C 180,E1 -5965.676,E2 -5965.676} C_VEL
LIN {X 0,Y 502.834,Z 377.853,A -85,B 0,C 180,E1 -5968.373,E2 -5968.373} C_VEL
LIN {X 0,Y 502.79,Z 377.857,A -85,B 0,C 180,E1 -5971.5,E2 -5971.5} C_VEL
LIN {X 0,Y 502.802,Z 377.856,A -85,B 0,C 180,E1 -5974.446,E2 -5974.446} C_VEL
LIN {X 0,Y 502.777,Z 377.858,A -85,B 0,C 180,E1 -5977.179,E2 -5977.179} C_VEL
LIN {X 0,Y 502.822,Z 377.853,A -85,B 0,C 180,E1 -5980.012,E2 -5980.012} C_VEL
LIN {X 0,Y 502.768,Z 377.858,A -85,B 0,C 180,E1 -5983.232,E2 -5983.232} C_VEL
LIN {X 0,Y 502.786,Z 377.857,A -85,B 0,C 180,E1 -5985.662,E2 -5985.662} C_VEL
LIN {X 0,Y 502.817,Z 377.854,A -85,B 0,C 180,E1 -5989.006,E2 -5989.006} C_VEL
LIN {X 0,Y 502.792,Z 377.857,A -85,B 0,C 180,E1 -5992.047,E2 -5992.047} C_VEL
LIN {X 0,Y 502.806,Z 377.854,A -85,B 0,C 180,E1 -5995.036,E2 -5995.036} C_VEL
LIN {X 0,Y 502.808,Z 377.853,A -85,B 0,C 180,E1 -5997.229,E2 -5997.229} C_VEL
LIN {X 0,Y 502.107,Z 377.943,A -85,B 0,C 180,E1 -5997.898,E2 -5997.898} C_VEL
LIN {X 0,Y 499.242,Z 378.299,A -85,B 0,C 180,E1 -5998.984,E2 -5998.984} C_VEL
LIN {X 0,Y 496.848,Z 378.597,A -85,B 0,C 180,E1 -5999.859,E2 -5999.859} C_VEL
LIN {X 0,Y 495.831,Z 378.723,A -85,B 0,C 180,E1 -6000.534,E2 -6000.534} C_VEL
LIN {X 0,Y 495.754,Z 378.732,A -85,B 0,C 180,E1 -6000.763,E2 -6000.763} C_VEL
LIN {X 0,Y 495.792,Z 378.729,A -85,B 0,C 180,E1 -6003.933,E2 -6003.933} C_VEL
LIN {X 0,Y 495.768,Z 378.732,A -85,B 0,C 180,E1 -6007.138,E2 -6007.138} C_VEL
LIN {X 0,Y 495.773,Z 378.733,A -85,B 0,C 180,E1 -6010.11,E2 -6010.11} C_VEL
LIN {X 0,Y 495.783,Z 378.728,A -85,B 0,C 180,E1 -6012.682,E2 -6012.682} C_VEL
LIN {X 0,Y 495.794,Z 378.728,A -85,B 0,C 180,E1 -6015.218,E2 -6015.218} C_VEL
LIN {X 0,Y 495.855,Z 378.72,A -85,B 0,C 180,E1 -6018.555,E2 -6018.555} C_VEL
LIN {X 0,Y 495.876,Z 378.719,A -85,B 0,C 180,E1 -6021.852,E2 -6021.852} C_VEL
LIN {X 0,Y 495.9,Z 378.716,A -85,B 0,C 180,E1 -6024.307,E2 -6024.307} C_VEL
LIN {X 0,Y 495.776,Z 378.734,A -85,B 0,C 180,E1 -6028.376,E2 -6028.376} C_VEL
LIN {X 0,Y 495.578,Z 378.898,A -85,B 0,C 180,E1 -6030,E2 -6030} C_VEL
LIN {X 0,Y 495.41,Z 383.269,A -85,B 0,C 180,E1 -6034.068,E2 -6034.068} C_VEL
LIN {X 0,Y 495.372,Z 386.166,A -85,B 0,C 180,E1 -6036.725,E2 -6036.725} C_VEL
LIN {X 0,Y 495.196,Z 389.536,A -85,B 0,C 180,E1 -6039.806,E2 -6039.806} C_VEL
LIN {X 0,Y 495.167,Z 392.247,A -85,B 0,C 180,E1 -6042.292,E2 -6042.292} C_VEL
LIN {X 0,Y 495.176,Z 395.455,A -85,B 0,C 180,E1 -6045.176,E2 -6045.176} C_VEL
LIN {X 0,Y 495.113,Z 398.29,A -85,B 0,C 180,E1 -6047.609,E2 -6047.609} C_VEL
LIN {X 0,Y 497.76,Z 410.83,A -85,B 0,C 180,E1 -6048.043,E2 -6048.043} C_VEL
LIN {X 0,Y 497.549,Z 422.287,A -85,B 0,C 180,E1 -6048.505,E2 -6048.505} C_VEL
LIN {X 0,Y 497.231,Z 433.097,A -85,B 0,C 180,E1 -6049.078,E2 -6049.078} C_VEL
LIN {X 0,Y 496.888,Z 444.379,A -85,B 0,C 180,E1 -6049.844,E2 -6049.844} C_VEL
LIN {X 0,Y 496.522,Z 454.661,A -85,B 0,C 180,E1 -6050.723,E2 -6050.723} C_VEL
LIN {X 0,Y 496.193,Z 463.169,A -85,B 0,C 180,E1 -6051.608,E2 -6051.608} C_VEL
LIN {X 0,Y 495.862,Z 471.711,A -85,B 0,C 180,E1 -6052.686,E2 -6052.686} C_VEL
LIN {X 0,Y 495.58,Z 479.185,A -85,B 0,C 180,E1 -6053.839,E2 -6053.839} C_VEL
LIN {X 0,Y 495.366,Z 486.181,A -85,B 0,C 180,E1 -6055.19,E2 -6055.19} C_VEL
LIN {X 0,Y 495.207,Z 491.816,A -85,B 0,C 180,E1 -6056.606,E2 -6056.606} C_VEL
LIN {X 0,Y 495.099,Z 495.772,A -85,B 0,C 180,E1 -6057.933,E2 -6057.933} C_VEL
LIN {X 0,Y 495.051,Z 497.85,A -85,B 0,C 180,E1 -6058.86,E2 -6058.86} C_VEL
LIN {X 0,Y 494.982,Z 499.626,A -85,B 0,C 180,E1 -6059.99,E2 -6059.99} C_VEL
LIN {X 0,Y 494.949,Z 500.389,A -85,B 0,C 180,E1 -6060.742,E2 -6060.742} C_VEL
LIN {X 0,Y 494.96,Z 500.832,A -85,B 0,C 180,E1 -6061.692,E2 -6061.692} C_VEL
LIN {X 0,Y 494.958,Z 500.554,A -85,B 0,C 180,E1 -6063.096,E2 -6063.096} C_VEL
LIN {X 0,Y 494.994,Z 498.968,A -85,B 0,C 180,E1 -6064.605,E2 -6064.605} C_VEL
LIN {X 0,Y 495.12,Z 496.25,A -85,B 0,C 180,E1 -6065.992,E2 -6065.992} C_VEL
LIN {X 0,Y 495.209,Z 492.295,A -85,B 0,C 180,E1 -6067.368,E2 -6067.368} C_VEL
LIN {X 0,Y 495.373,Z 487.105,A -85,B 0,C 180,E1 -6068.711,E2 -6068.711} C_VEL
LIN {X 0,Y 495.56,Z 480.634,A -85,B 0,C 180,E1 -6070.019,E2 -6070.019} C_VEL
LIN {X 0,Y 495.841,Z 472.581,A -85,B 0,C 180,E1 -6071.304,E2 -6071.304} C_VEL
LIN {X 0,Y 496.243,Z 463.212,A -85,B 0,C 180,E1 -6072.495,E2 -6072.495} C_VEL
LIN {X 0,Y 496.527,Z 453.799,A -85,B 0,C 180,E1 -6073.469,E2 -6073.469} C_VEL
LIN {X 0,Y 496.858,Z 443.917,A -85,B 0,C 180,E1 -6074.298,E2 -6074.298} C_VEL
LIN {X 0,Y 497.269,Z 432.174,A -85,B 0,C 180,E1 -6075.079,E2 -6075.079} C_VEL
LIN {X 0,Y 497.587,Z 420.235,A -85,B 0,C 180,E1 -6075.691,E2 -6075.691} C_VEL
LIN {X 0,Y 497.626,Z 410.334,A -85,B 0,C 180,E1 -6076.076,E2 -6076.076} C_VEL
LIN {X 0,Y 495.459,Z 400.389,A -85,B 0,C 180,E1 -6076.427,E2 -6076.427} C_VEL
LIN {X 0,Y 495.058,Z 398.536,A -85,B 0,C 180,E1 -6076.486,E2 -6076.486} C_VEL
LIN {X 0,Y 495.096,Z 395.536,A -85,B 0,C 180,E1 -6079.233,E2 -6079.233} C_VEL
LIN {X 0,Y 495.103,Z 392.164,A -85,B 0,C 180,E1 -6082.382,E2 -6082.382} C_VEL
LIN {X 0,Y 495.248,Z 388.916,A -85,B 0,C 180,E1 -6085.414,E2 -6085.414} C_VEL
LIN {X 0,Y 495.341,Z 385.819,A -85,B 0,C 180,E1 -6088.351,E2 -6088.351} C_VEL
LIN {X 0,Y 495.353,Z 382.865,A -85,B 0,C 180,E1 -6091.158,E2 -6091.158} C_VEL
LIN {X 0,Y 495.377,Z 379.93,A -85,B 0,C 180,E1 -6093.908,E2 -6093.908} C_VEL
LIN {X 0,Y 495.479,Z 378.77,A -85,B 0,C 180,E1 -6095.2,E2 -6095.2} C_VEL
LIN {X 0,Y 495.713,Z 378.742,A -85,B 0,C 180,E1 -6097.493,E2 -6097.493} C_VEL
LIN {X 0,Y 495.773,Z 378.732,A -85,B 0,C 180,E1 -6100.11,E2 -6100.11} C_VEL
LIN {X 0,Y 495.781,Z 378.729,A -85,B 0,C 180,E1 -6102.681,E2 -6102.681} C_VEL
LIN {X 0,Y 495.784,Z 378.729,A -85,B 0,C 180,E1 -6105.217,E2 -6105.217} C_VEL
LIN {X 0,Y 495.849,Z 378.721,A -85,B 0,C 180,E1 -6108.555,E2 -6108.555} C_VEL
LIN {X 0,Y 495.867,Z 378.721,A -85,B 0,C 180,E1 -6111.852,E2 -6111.852} C_VEL
LIN {X 0,Y 495.89,Z 378.717,A -85,B 0,C 180,E1 -6114.306,E2 -6114.306} C_VEL
LIN {X 0,Y 495.988,Z 378.703,A -85,B 0,C 180,E1 -6117.564,E2 -6117.564} C_VEL
LIN {X 0,Y 495.99,Z 378.702,A -85,B 0,C 180,E1 -6120,E2 -6120} C_VEL
LIN {X 0,Y 495.986,Z 378.703,A -85,B 0,C 180,E1 -6122.436,E2 -6122.436} C_VEL
LIN {X 0,Y 495.888,Z 378.715,A -85,B 0,C 180,E1 -6125.693,E2 -6125.693} C_VEL
LIN {X 0,Y 495.867,Z 378.717,A -85,B 0,C 180,E1 -6128.148,E2 -6128.148} C_VEL
LIN {X 0,Y 495.849,Z 378.722,A -85,B 0,C 180,E1 -6131.445,E2 -6131.445} C_VEL
LIN {X 0,Y 495.784,Z 378.731,A -85,B 0,C 180,E1 -6134.783,E2 -6134.783} C_VEL
LIN {X 0,Y 495.782,Z 378.732,A -85,B 0,C 180,E1 -6137.319,E2 -6137.319} C_VEL
LIN {X 0,Y 495.766,Z 378.733,A -85,B 0,C 180,E1 -6139.891,E2 -6139.891} C_VEL
LIN {X 0,Y 495.756,Z 378.733,A -85,B 0,C 180,E1 -6142.862,E2 -6142.862} C_VEL
LIN {X 0,Y 495.794,Z 378.727,A -85,B 0,C 180,E1 -6146.068,E2 -6146.068} C_VEL
LIN {X 0,Y 495.767,Z 378.73,A -85,B 0,C 180,E1 -6148.815,E2 -6148.815} C_VEL
LIN {X 0,Y 495.75,Z 378.736,A -85,B 0,C 180,E1 -6151.726,E2 -6151.726} C_VEL
LIN {X 0,Y 495.758,Z 378.734,A -85,B 0,C 180,E1 -6154.693,E2 -6154.693} C_VEL
LIN {X 0,Y 495.727,Z 378.738,A -85,B 0,C 180,E1 -6157.562,E2 -6157.562} C_VEL
LIN {X 0,Y 495.79,Z 378.731,A -85,B 0,C 180,E1 -6160.052,E2 -6160.052} C_VEL
LIN {X 0,Y 495.722,Z 378.738,A -85,B 0,C 180,E1 -6162.884,E2 -6162.884} C_VEL
LIN {X 0,Y 495.732,Z 378.738,A -85,B 0,C 180,E1 -6166,E2 -6166} C_VEL
LIN {X 0,Y 495.775,Z 378.734,A -85,B 0,C 180,E1 -6169.302,E2 -6169.302} C_VEL
LIN {X 0,Y 495.774,Z 378.799,A -85,B 0,C 180,E1 -6170.364,E2 -6170.364} C_VEL
LIN {X 0,Y 497.195,Z 386.391,A -85,B 0,C 180,E1 -6173.582,E2 -6173.582} C_VEL
LIN {X 0,Y 497.16,Z 391.654,A -85,B 0,C 180,E1 -6175.567,E2 -6175.567} C_VEL
LIN {X 0,Y 496.806,Z 399.463,A -85,B 0,C 180,E1 -6178.439,E2 -6178.439} C_VEL
LIN {X 0,Y 496.51,Z 409.181,A -85,B 0,C 180,E1 -6181.753,E2 -6181.753} C_VEL
LIN {X 0,Y 496.259,Z 417.043,A -85,B 0,C 180,E1 -6184.41,E2 -6184.41} C_VEL
LIN {X 0,Y 496.019,Z 426.818,A -85,B 0,C 180,E1 -6187.508,E2 -6187.508} C_VEL
LIN {X 0,Y 495.774,Z 436.14,A -85,B 0,C 180,E1 -6190.541,E2 -6190.541} C_VEL
LIN {X 0,Y 495.549,Z 445.408,A -85,B 0,C 180,E1 -6193.522,E2 -6193.522} C_VEL
LIN {X 0,Y 495.418,Z 451.582,A -85,B 0,C 180,E1 -6195.485,E2 -6195.485} C_VEL
LIN {X 0,Y 497.582,Z 464.642,A -85,B 0,C 180,E1 -6195.859,E2 -6195.859} C_VEL
LIN {X 0,Y 497.573,Z 475.774,A -85,B 0,C 180,E1 -6196.263,E2 -6196.263} C_VEL
LIN {X 0,Y 497.224,Z 487.409,A -85,B 0,C 180,E1 -6196.826,E2 -6196.826} C_VEL
LIN {X 0,Y 496.798,Z 499.137,A -85,B 0,C 180,E1 -6197.57,E2 -6197.57} C_VEL
LIN {X 0,Y 496.471,Z 510.265,A -85,B 0,C 180,E1 -6198.466,E2 -6198.466} C_VEL
LIN {X 0,Y 496.069,Z 519.539,A -85,B 0,C 180,E1 -6199.387,E2 -6199.387} C_VEL
LIN {X 0,Y 495.791,Z 527.991,A -85,B 0,C 180,E1 -6200.412,E2 -6200.412} C_VEL
LIN {X 0,Y 495.485,Z 536.236,A -85,B 0,C 180,E1 -6201.64,E2 -6201.64} C_VEL
LIN {X 0,Y 495.261,Z 542.876,A -85,B 0,C 180,E1 -6202.868,E2 -6202.868} C_VEL
LIN {X 0,Y 495.178,Z 548.949,A -85,B 0,C 180,E1 -6204.298,E2 -6204.298} C_VEL
LIN {X 0,Y 495.029,Z 552.894,A -85,B 0,C 180,E1 -6205.521,E2 -6205.521} C_VEL
LIN {X 0,Y 495.043,Z 555.807,A -85,B 0,C 180,E1 -6206.744,E2 -6206.744} C_VEL
LIN {X 0,Y 494.961,Z 558.183,A -85,B 0,C 180,E1 -6208.373,E2 -6208.373} C_VEL
LIN {X 0,Y 494.898,Z 559,A -85,B 0,C 180,E1 -6210,E2 -6210} C_VEL
LIN {X 0,Y 494.961,Z 558.185,A -85,B 0,C 180,E1 -6211.627,E2 -6211.627} C_VEL
LIN {X 0,Y 495.043,Z 555.81,A -85,B 0,C 180,E1 -6213.255,E2 -6213.255} C_VEL
LIN {X 0,Y 495.029,Z 552.896,A -85,B 0,C 180,E1 -6214.478,E2 -6214.478} C_VEL
LIN {X 0,Y 495.208,Z 547.805,A -85,B 0,C 180,E1 -6215.999,E2 -6215.999} C_VEL
LIN {X 0,Y 495.277,Z 541.871,A -85,B 0,C 180,E1 -6217.337,E2 -6217.337} C_VEL
LIN {X 0,Y 495.557,Z 535.005,A -85,B 0,C 180,E1 -6218.563,E2 -6218.563} C_VEL
LIN {X 0,Y 495.852,Z 526.416,A -85,B 0,C 180,E1 -6219.792,E2 -6219.792} C_VEL
LIN {X 0,Y 496.209,Z 517.602,A -85,B 0,C 180,E1 -6220.816,E2 -6220.816} C_VEL
LIN {X 0,Y 496.589,Z 506.75,A -85,B 0,C 180,E1 -6221.841,E2 -6221.841} C_VEL
LIN {X 0,Y 496.895,Z 496.787,A -85,B 0,C 180,E1 -6222.597,E2 -6222.597} C_VEL
LIN {X 0,Y 497.232,Z 485.498,A -85,B 0,C 180,E1 -6223.278,E2 -6223.278} C_VEL
LIN {X 0,Y 497.64,Z 473.178,A -85,B 0,C 180,E1 -6223.839,E2 -6223.839} C_VEL
LIN {X 0,Y 497.59,Z 464.648,A -85,B 0,C 180,E1 -6224.14,E2 -6224.14} C_VEL
LIN {X 0,Y 495.427,Z 451.532,A -85,B 0,C 180,E1 -6224.531,E2 -6224.531} C_VEL
LIN {X 0,Y 495.637,Z 441.437,A -85,B 0,C 180,E1 -6227.749,E2 -6227.749} C_VEL
LIN {X 0,Y 495.884,Z 432.17,A -85,B 0,C 180,E1 -6230.751,E2 -6230.751} C_VEL
LIN {X 0,Y 496.102,Z 422.683,A -85,B 0,C 180,E1 -6233.812,E2 -6233.812} C_VEL
LIN {X 0,Y 496.34,Z 414.566,A -85,B 0,C 180,E1 -6236.455,E2 -6236.455} C_VEL
LIN {X 0,Y 496.586,Z 406.551,A -85,B 0,C 180,E1 -6239.226,E2 -6239.226} C_VEL
LIN {X 0,Y 496.912,Z 398.852,A -85,B 0,C 180,E1 -6241.94,E2 -6241.94} C_VEL
LIN {X 0,Y 497.268,Z 390.548,A -85,B 0,C 180,E1 -6244.942,E2 -6244.942} C_VEL
LIN {X 0,Y 497.185,Z 386.619,A -85,B 0,C 180,E1 -6246.418,E2 -6246.418} C_VEL
LIN {X 0,Y 496.151,Z 380.785,A -85,B 0,C 180,E1 -6248.824,E2 -6248.824} C_VEL
LIN {X 0,Y 495.76,Z 378.734,A -85,B 0,C 180,E1 -6249.738,E2 -6249.738} C_VEL
LIN {X 0,Y 495.722,Z 378.74,A -85,B 0,C 180,E1 -6252.882,E2 -6252.882} C_VEL
LIN {X 0,Y 495.729,Z 378.738,A -85,B 0,C 180,E1 -6255.998,E2 -6255.998} C_VEL
LIN {X 0,Y 495.775,Z 378.732,A -85,B 0,C 180,E1 -6259.301,E2 -6259.301} C_VEL
LIN {X 0,Y 495.725,Z 378.736,A -85,B 0,C 180,E1 -6262.438,E2 -6262.438} C_VEL
LIN {X 0,Y 495.779,Z 378.73,A -85,B 0,C 180,E1 -6265.457,E2 -6265.457} C_VEL
LIN {X 0,Y 495.752,Z 378.734,A -85,B 0,C 180,E1 -6268.363,E2 -6268.363} C_VEL
LIN {X 0,Y 495.78,Z 378.731,A -85,B 0,C 180,E1 -6271.506,E2 -6271.506} C_VEL
LIN {X 0,Y 495.791,Z 378.728,A -85,B 0,C 180,E1 -6273.932,E2 -6273.932} C_VEL
LIN {X 0,Y 495.749,Z 378.736,A -85,B 0,C 180,E1 -6277.139,E2 -6277.139} C_VEL
LIN {X 0,Y 495.77,Z 378.73,A -85,B 0,C 180,E1 -6280.11,E2 -6280.11} C_VEL
LIN {X 0,Y 495.779,Z 378.732,A -85,B 0,C 180,E1 -6282.681,E2 -6282.681} C_VEL
LIN {X 0,Y 495.78,Z 378.73,A -85,B 0,C 180,E1 -6285.217,E2 -6285.217} C_VEL
LIN {X 0,Y 495.846,Z 378.723,A -85,B 0,C 180,E1 -6288.555,E2 -6288.555} C_VEL
LIN {X 0,Y 495.864,Z 378.72,A -85,B 0,C 180,E1 -6291.852,E2 -6291.852} C_VEL
LIN {X 0,Y 495.886,Z 378.717,A -85,B 0,C 180,E1 -6294.306,E2 -6294.306} C_VEL
LIN {X 0,Y 495.984,Z 378.703,A -85,B 0,C 180,E1 -6297.564,E2 -6297.564} C_VEL
LIN {X 0,Y 495.987,Z 378.703,A -85,B 0,C 180,E1 -6300,E2 -6300} C_VEL
LIN {X 0,Y 495.984,Z 378.705,A -85,B 0,C 180,E1 -6302.436,E2 -6302.436} C_VEL
LIN {X 0,Y 495.887,Z 378.715,A -85,B 0,C 180,E1 -6305.694,E2 -6305.694} C_VEL
LIN {X 0,Y 495.865,Z 378.72,A -85,B 0,C 180,E1 -6308.148,E2 -6308.148} C_VEL
LIN {X 0,Y 495.846,Z 378.722,A -85,B 0,C 180,E1 -6311.445,E2 -6311.445} C_VEL
LIN {X 0,Y 495.781,Z 378.732,A -85,B 0,C 180,E1 -6314.783,E2 -6314.783} C_VEL
LIN {X 0,Y 495.779,Z 378.729,A -85,B 0,C 180,E1 -6317.319,E2 -6317.319} C_VEL
LIN {X 0,Y 495.77,Z 378.731,A -85,B 0,C 180,E1 -6319.891,E2 -6319.891} C_VEL
LIN {X 0,Y 495.75,Z 378.734,A -85,B 0,C 180,E1 -6322.861,E2 -6322.861} C_VEL
LIN {X 0,Y 495.792,Z 378.731,A -85,B 0,C 180,E1 -6326.068,E2 -6326.068} C_VEL
LIN {X 0,Y 495.765,Z 378.732,A -85,B 0,C 180,E1 -6328.815,E2 -6328.815} C_VEL
LIN {X 0,Y 495.752,Z 378.735,A -85,B 0,C 180,E1 -6331.727,E2 -6331.727} C_VEL
LIN {X 0,Y 495.772,Z 378.732,A -85,B 0,C 180,E1 -6334.696,E2 -6334.696} C_VEL
LIN {X 0,Y 495.728,Z 378.736,A -85,B 0,C 180,E1 -6337.562,E2 -6337.562} C_VEL
LIN {X 0,Y 495.789,Z 378.73,A -85,B 0,C 180,E1 -6340.053,E2 -6340.053} C_VEL
LIN {X 0,Y 495.721,Z 378.736,A -85,B 0,C 180,E1 -6342.884,E2 -6342.884} C_VEL
LIN {X 0,Y 495.731,Z 378.738,A -85,B 0,C 180,E1 -6346,E2 -6346} C_VEL
LIN {X 0,Y 495.764,Z 378.732,A -85,B 0,C 180,E1 -6349.301,E2 -6349.301} C_VEL
LIN {X 0,Y 495.729,Z 378.738,A -85,B 0,C 180,E1 -6352.44,E2 -6352.44} C_VEL
LIN {X 0,Y 495.782,Z 378.729,A -85,B 0,C 180,E1 -6355.458,E2 -6355.458} C_VEL
LIN {X 0,Y 495.756,Z 378.733,A -85,B 0,C 180,E1 -6358.365,E2 -6358.365} C_VEL
LIN {X 0,Y 495.754,Z 378.732,A -85,B 0,C 180,E1 -6360.763,E2 -6360.763} C_VEL
LIN {X 0,Y 495.097,Z 378.816,A -85,B 0,C 180,E1 -6361.442,E2 -6361.442} C_VEL
LIN {X 0,Y 492.24,Z 379.171,A -85,B 0,C 180,E1 -6362.545,E2 -6362.545} C_VEL
LIN {X 0,Y 489.832,Z 379.47,A -85,B 0,C 180,E1 -6363.433,E2 -6363.433} C_VEL
LIN {X 0,Y 488.816,Z 379.598,A -85,B 0,C 180,E1 -6364.12,E2 -6364.12} C_VEL
LIN {X 0,Y 488.744,Z 379.607,A -85,B 0,C 180,E1 -6364.352,E2 -6364.352} C_VEL
LIN {X 0,Y 488.73,Z 379.608,A -85,B 0,C 180,E1 -6367.154,E2 -6367.154} C_VEL
LIN {X 0,Y 488.727,Z 379.609,A -85,B 0,C 180,E1 -6369.811,E2 -6369.811} C_VEL
LIN {X 0,Y 488.731,Z 379.608,A -85,B 0,C 180,E1 -6372.424,E2 -6372.424} C_VEL
LIN {X 0,Y 488.765,Z 379.603,A -85,B 0,C 180,E1 -6375,E2 -6375} C_VEL
LIN {X 0,Y 488.809,Z 379.598,A -85,B 0,C 180,E1 -6378.388,E2 -6378.388} C_VEL
LIN {X 0,Y 488.82,Z 379.598,A -85,B 0,C 180,E1 -6381.734,E2 -6381.734} C_VEL
LIN {X 0,Y 488.859,Z 379.593,A -85,B 0,C 180,E1 -6384.225,E2 -6384.225} C_VEL
LIN {X 0,Y 488.749,Z 379.609,A -85,B 0,C 180,E1 -6388.352,E2 -6388.352} C_VEL
LIN {X 0,Y 488.529,Z 379.636,A -85,B 0,C 180,E1 -6390,E2 -6390} C_VEL
LIN {X 0,Y 488.367,Z 384.042,A -85,B 0,C 180,E1 -6394.126,E2 -6394.126} C_VEL
LIN {X 0,Y 488.317,Z 386.864,A -85,B 0,C 180,E1 -6396.747,E2 -6396.747} C_VEL
LIN {X 0,Y 488.125,Z 390.34,A -85,B 0,C 180,E1 -6399.949,E2 -6399.949} C_VEL
LIN {X 0,Y 488.086,Z 393.099,A -85,B 0,C 180,E1 -6402.473,E2 -6402.473} C_VEL
LIN {X 0,Y 488.083,Z 396.13,A -85,B 0,C 180,E1 -6405.258,E2 -6405.258} C_VEL
LIN {X 0,Y 488.03,Z 398.536,A -85,B 0,C 180,E1 -6407.386,E2 -6407.386} C_VEL
LIN {X 0,Y 490.914,Z 411.995,A -85,B 0,C 180,E1 -6407.873,E2 -6407.873} C_VEL
LIN {X 0,Y 490.594,Z 424.905,A -85,B 0,C 180,E1 -6408.417,E2 -6408.417} C_VEL
LIN {X 0,Y 490.205,Z 437.396,A -85,B 0,C 180,E1 -6409.142,E2 -6409.142} C_VEL
LIN {X 0,Y 489.889,Z 447.867,A -85,B 0,C 180,E1 -6409.921,E2 -6409.921} C_VEL
LIN {X 0,Y 489.481,Z 457.556,A -85,B 0,C 180,E1 -6410.805,E2 -6410.805} C_VEL
LIN {X 0,Y 489.144,Z 465.75,A -85,B 0,C 180,E1 -6411.714,E2 -6411.714} C_VEL
LIN {X 0,Y 488.793,Z 474.154,A -85,B 0,C 180,E1 -6412.843,E2 -6412.843} C_VEL
LIN {X 0,Y 488.524,Z 481.052,A -85,B 0,C 180,E1 -6413.979,E2 -6413.979} C_VEL
LIN {X 0,Y 488.293,Z 487.182,A -85,B 0,C 180,E1 -6415.225,E2 -6415.225} C_VEL
LIN {X 0,Y 488.164,Z 492.163,A -85,B 0,C 180,E1 -6416.506,E2 -6416.506} C_VEL
LIN {X 0,Y 488.035,Z 496.28,A -85,B 0,C 180,E1 -6417.905,E2 -6417.905} C_VEL
LIN {X 0,Y 487.928,Z 499.166,A -85,B 0,C 180,E1 -6419.322,E2 -6419.322} C_VEL
LIN {X 0,Y 487.876,Z 500.396,A -85,B 0,C 180,E1 -6420.277,E2 -6420.277} C_VEL
LIN {X 0,Y 487.867,Z 501.288,A -85,B 0,C 180,E1 -6421.796,E2 -6421.796} C_VEL
LIN {X 0,Y 487.867,Z 500.867,A -85,B 0,C 180,E1 -6423.329,E2 -6423.329} C_VEL
LIN {X 0,Y 487.926,Z 499.13,A -85,B 0,C 180,E1 -6424.813,E2 -6424.813} C_VEL
LIN {X 0,Y 488.047,Z 496.175,A -85,B 0,C 180,E1 -6426.252,E2 -6426.252} C_VEL
LIN {X 0,Y 488.181,Z 492.05,A -85,B 0,C 180,E1 -6427.646,E2 -6427.646} C_VEL
LIN {X 0,Y 488.364,Z 486.702,A -85,B 0,C 180,E1 -6429.003,E2 -6429.003} C_VEL
LIN {X 0,Y 488.597,Z 479.935,A -85,B 0,C 180,E1 -6430.336,E2 -6430.336} C_VEL
LIN {X 0,Y 488.886,Z 471.703,A -85,B 0,C 180,E1 -6431.623,E2 -6431.623} C_VEL
LIN {X 0,Y 489.264,Z 463.297,A -85,B 0,C 180,E1 -6432.687,E2 -6432.687} C_VEL
LIN {X 0,Y 489.614,Z 453.401,A -85,B 0,C 180,E1 -6433.709,E2 -6433.709} C_VEL
LIN {X 0,Y 490.064,Z 442.008,A -85,B 0,C 180,E1 -6434.644,E2 -6434.644} C_VEL
LIN {X 0,Y 490.477,Z 430.26,A -85,B 0,C 180,E1 -6435.403,E2 -6435.403} C_VEL
LIN {X 0,Y 490.774,Z 419.03,A -85,B 0,C 180,E1 -6435.957,E2 -6435.957} C_VEL
LIN {X 0,Y 490.723,Z 410.989,A -85,B 0,C 180,E1 -6436.269,E2 -6436.269} C_VEL
LIN {X 0,Y 487.98,Z 398.987,A -85,B 0,C 180,E1 -6436.698,E2 -6436.698} C_VEL
LIN {X 0,Y 488.032,Z 395.684,A -85,B 0,C 180,E1 -6439.749,E2 -6439.749} C_VEL
LIN {X 0,Y 488.048,Z 392.457,A -85,B 0,C 180,E1 -6442.785,E2 -6442.785} C_VEL
LIN {X 0,Y 488.177,Z 389.192,A -85,B 0,C 180,E1 -6445.843,E2 -6445.843} C_VEL
LIN {X 0,Y 488.278,Z 386.125,A -85,B 0,C 180,E1 -6448.791,E2 -6448.791} C_VEL
LIN {X 0,Y 488.315,Z 383.114,A -85,B 0,C 180,E1 -6451.644,E2 -6451.644} C_VEL
LIN {X 0,Y 488.357,Z 380.194,A -85,B 0,C 180,E1 -6454.422,E2 -6454.422} C_VEL
LIN {X 0,Y 488.442,Z 379.647,A -85,B 0,C 180,E1 -6455.337,E2 -6455.337} C_VEL
LIN {X 0,Y 488.679,Z 379.617,A -85,B 0,C 180,E1 -6458.042,E2 -6458.042} C_VEL
LIN {X 0,Y 488.741,Z 379.608,A -85,B 0,C 180,E1 -6460.686,E2 -6460.686} C_VEL
LIN {X 0,Y 488.725,Z 379.611,A -85,B 0,C 180,E1 -6463.285,E2 -6463.285} C_VEL
LIN {X 0,Y 488.732,Z 379.611,A -85,B 0,C 180,E1 -6465.85,E2 -6465.85} C_VEL
LIN {X 0,Y 488.802,Z 379.6,A -85,B 0,C 180,E1 -6468.387,E2 -6468.387} C_VEL
LIN {X 0,Y 488.812,Z 379.6,A -85,B 0,C 180,E1 -6471.733,E2 -6471.733} C_VEL
LIN {X 0,Y 488.85,Z 379.595,A -85,B 0,C 180,E1 -6474.224,E2 -6474.224} C_VEL
LIN {X 0,Y 488.956,Z 379.578,A -85,B 0,C 180,E1 -6477.529,E2 -6477.529} C_VEL
LIN {X 0,Y 488.97,Z 379.578,A -85,B 0,C 180,E1 -6480.823,E2 -6480.823} C_VEL
LIN {X 0,Y 488.954,Z 379.58,A -85,B 0,C 180,E1 -6482.471,E2 -6482.471} C_VEL
LIN {X 0,Y 488.848,Z 379.592,A -85,B 0,C 180,E1 -6485.776,E2 -6485.776} C_VEL
LIN {X 0,Y 488.811,Z 379.596,A -85,B 0,C 180,E1 -6488.266,E2 -6488.266} C_VEL
LIN {X 0,Y 488.802,Z 379.599,A -85,B 0,C 180,E1 -6491.612,E2 -6491.612} C_VEL
LIN {X 0,Y 488.756,Z 379.606,A -85,B 0,C 180,E1 -6495.001,E2 -6495.001} C_VEL
LIN {X 0,Y 488.749,Z 379.606,A -85,B 0,C 180,E1 -6498.442,E2 -6498.442} C_VEL
LIN {X 0,Y 488.701,Z 379.613,A -85,B 0,C 180,E1 -6501.071,E2 -6501.071} C_VEL
LIN {X 0,Y 488.687,Z 379.613,A -85,B 0,C 180,E1 -6503.746,E2 -6503.746} C_VEL
LIN {X 0,Y 488.794,Z 379.601,A -85,B 0,C 180,E1 -6506.946,E2 -6506.946} C_VEL
LIN {X 0,Y 488.704,Z 379.613,A -85,B 0,C 180,E1 -6510.363,E2 -6510.363} C_VEL
LIN {X 0,Y 488.724,Z 379.61,A -85,B 0,C 180,E1 -6513.484,E2 -6513.484} C_VEL
LIN {X 0,Y 488.678,Z 379.617,A -85,B 0,C 180,E1 -6516.355,E2 -6516.355} C_VEL
LIN {X 0,Y 488.746,Z 379.609,A -85,B 0,C 180,E1 -6519.25,E2 -6519.25} C_VEL
LIN {X 0,Y 488.688,Z 379.615,A -85,B 0,C 180,E1 -6522.526,E2 -6522.526} C_VEL
LIN {X 0,Y 488.709,Z 379.614,A -85,B 0,C 180,E1 -6525.199,E2 -6525.199} C_VEL
LIN {X 0,Y 488.708,Z 379.614,A -85,B 0,C 180,E1 -6528.4,E2 -6528.4} C_VEL
LIN {X 0,Y 488.754,Z 379.715,A -85,B 0,C 180,E1 -6530.083,E2 -6530.083} C_VEL
LIN {X 0,Y 490.162,Z 387.391,A -85,B 0,C 180,E1 -6533.411,E2 -6533.411} C_VEL
LIN {X 0,Y 490.239,Z 391.415,A -85,B 0,C 180,E1 -6535.011,E2 -6535.011} C_VEL
LIN {X 0,Y 489.882,Z 399.388,A -85,B 0,C 180,E1 -6537.94,E2 -6537.94} C_VEL
LIN {X 0,Y 489.517,Z 407.398,A -85,B 0,C 180,E1 -6540.782,E2 -6540.782} C_VEL
LIN {X 0,Y 489.288,Z 415.442,A -85,B 0,C 180,E1 -6543.559,E2 -6543.559} C_VEL
LIN {X 0,Y 489.044,Z 423.668,A -85,B 0,C 180,E1 -6546.273,E2 -6546.273} C_VEL
LIN {X 0,Y 488.828,Z 433.73,A -85,B 0,C 180,E1 -6549.48,E2 -6549.48} C_VEL
LIN {X 0,Y 488.582,Z 442.76,A -85,B 0,C 180,E1 -6552.418,E2 -6552.418} C_VEL
LIN {X 0,Y 488.375,Z 451.582,A -85,B 0,C 180,E1 -6555.271,E2 -6555.271} C_VEL
LIN {X 0,Y 490.635,Z 465.098,A -85,B 0,C 180,E1 -6555.668,E2 -6555.668} C_VEL
LIN {X 0,Y 490.747,Z 473.176,A -85,B 0,C 180,E1 -6555.962,E2 -6555.962} C_VEL
LIN {X 0,Y 490.32,Z 485.491,A -85,B 0,C 180,E1 -6556.531,E2 -6556.531} C_VEL
LIN {X 0,Y 489.964,Z 497.01,A -85,B 0,C 180,E1 -6557.237,E2 -6557.237} C_VEL
LIN {X 0,Y 489.599,Z 507.92,A -85,B 0,C 180,E1 -6558.092,E2 -6558.092} C_VEL
LIN {X 0,Y 489.175,Z 517.598,A -85,B 0,C 180,E1 -6559.026,E2 -6559.026} C_VEL
LIN {X 0,Y 488.847,Z 526.412,A -85,B 0,C 180,E1 -6560.066,E2 -6560.066} C_VEL
LIN {X 0,Y 488.509,Z 535.003,A -85,B 0,C 180,E1 -6561.312,E2 -6561.312} C_VEL
LIN {X 0,Y 488.207,Z 541.868,A -85,B 0,C 180,E1 -6562.556,E2 -6562.556} C_VEL
LIN {X 0,Y 488.096,Z 547.062,A -85,B 0,C 180,E1 -6563.722,E2 -6563.722} C_VEL
LIN {X 0,Y 487.971,Z 551.676,A -85,B 0,C 180,E1 -6565.043,E2 -6565.043} C_VEL
LIN {X 0,Y 487.947,Z 553.958,A -85,B 0,C 180,E1 -6565.87,E2 -6565.87} C_VEL
LIN {X 0,Y 487.967,Z 555.807,A -85,B 0,C 180,E1 -6566.697,E2 -6566.697} C_VEL
LIN {X 0,Y 487.889,Z 558.183,A -85,B 0,C 180,E1 -6568.349,E2 -6568.349} C_VEL
LIN {X 0,Y 487.819,Z 559,A -85,B 0,C 180,E1 -6570,E2 -6570} C_VEL
LIN {X 0,Y 487.889,Z 558.184,A -85,B 0,C 180,E1 -6571.651,E2 -6571.651} C_VEL
LIN {X 0,Y 487.966,Z 555.81,A -85,B 0,C 180,E1 -6573.302,E2 -6573.302} C_VEL
LIN {X 0,Y 487.938,Z 552.896,A -85,B 0,C 180,E1 -6574.543,E2 -6574.543} C_VEL
LIN {X 0,Y 488.104,Z 548.949,A -85,B 0,C 180,E1 -6575.784,E2 -6575.784} C_VEL
LIN {X 0,Y 488.19,Z 542.877,A -85,B 0,C 180,E1 -6577.236,E2 -6577.236} C_VEL
LIN {X 0,Y 488.453,Z 536.238,A -85,B 0,C 180,E1 -6578.481,E2 -6578.481} C_VEL
LIN {X 0,Y 488.764,Z 527.995,A -85,B 0,C 180,E1 -6579.727,E2 -6579.727} C_VEL
LIN {X 0,Y 489.095,Z 519.543,A -85,B 0,C 180,E1 -6580.766,E2 -6580.766} C_VEL
LIN {X 0,Y 489.585,Z 509.097,A -85,B 0,C 180,E1 -6581.803,E2 -6581.803} C_VEL
LIN {X 0,Y 489.926,Z 497.639,A -85,B 0,C 180,E1 -6582.718,E2 -6582.718} C_VEL
LIN {X 0,Y 490.265,Z 487.413,A -85,B 0,C 180,E1 -6583.365,E2 -6583.365} C_VEL
LIN {X 0,Y 490.648,Z 475.776,A -85,B 0,C 180,E1 -6583.935,E2 -6583.935} C_VEL
LIN {X 0,Y 490.707,Z 465.535,A -85,B 0,C 180,E1 -6584.316,E2 -6584.316} C_VEL
LIN {X 0,Y 488.499,Z 452.509,A -85,B 0,C 180,E1 -6584.708,E2 -6584.708} C_VEL
LIN {X 0,Y 488.383,Z 451.532,A -85,B 0,C 180,E1 -6584.745,E2 -6584.745} C_VEL
LIN {X 0,Y 488.61,Z 441.614,A -85,B 0,C 180,E1 -6587.955,E2 -6587.955} C_VEL
LIN {X 0,Y 488.859,Z 432.04,A -85,B 0,C 180,E1 -6591.063,E2 -6591.063} C_VEL
LIN {X 0,Y 489.071,Z 422.385,A -85,B 0,C 180,E1 -6594.176,E2 -6594.176} C_VEL
LIN {X 0,Y 489.296,Z 415.587,A -85,B 0,C 180,E1 -6596.44,E2 -6596.44} C_VEL
LIN {X 0,Y 489.559,Z 407.671,A -85,B 0,C 180,E1 -6599.215,E2 -6599.215} C_VEL
LIN {X 0,Y 489.939,Z 399.37,A -85,B 0,C 180,E1 -6602.185,E2 -6602.185} C_VEL
LIN {X 0,Y 490.32,Z 391.14,A -85,B 0,C 180,E1 -6605.213,E2 -6605.213} C_VEL
LIN {X 0,Y 490.2,Z 387.622,A -85,B 0,C 180,E1 -6606.595,E2 -6606.595} C_VEL
LIN {X 0,Y 489.042,Z 381.391,A -85,B 0,C 180,E1 -6609.22,E2 -6609.22} C_VEL
LIN {X 0,Y 488.734,Z 379.607,A -85,B 0,C 180,E1 -6610.052,E2 -6610.052} C_VEL
LIN {X 0,Y 488.705,Z 379.613,A -85,B 0,C 180,E1 -6612.826,E2 -6612.826} C_VEL
LIN {X 0,Y 488.694,Z 379.614,A -85,B 0,C 180,E1 -6615.975,E2 -6615.975} C_VEL
LIN {X 0,Y 488.708,Z 379.613,A -85,B 0,C 180,E1 -6618.584,E2 -6618.584} C_VEL
LIN {X 0,Y 488.739,Z 379.608,A -85,B 0,C 180,E1 -6620.941,E2 -6620.941} C_VEL
LIN {X 0,Y 488.679,Z 379.614,A -85,B 0,C 180,E1 -6623.868,E2 -6623.868} C_VEL
LIN {X 0,Y 488.733,Z 379.608,A -85,B 0,C 180,E1 -6626.877,E2 -6626.877} C_VEL
LIN {X 0,Y 488.716,Z 379.609,A -85,B 0,C 180,E1 -6629.78,E2 -6629.78} C_VEL
LIN {X 0,Y 488.791,Z 379.601,A -85,B 0,C 180,E1 -6633.054,E2 -6633.054} C_VEL
LIN {X 0,Y 488.685,Z 379.614,A -85,B 0,C 180,E1 -6636.254,E2 -6636.254} C_VEL
LIN {X 0,Y 488.737,Z 379.608,A -85,B 0,C 180,E1 -6639.175,E2 -6639.175} C_VEL
LIN {X 0,Y 488.75,Z 379.606,A -85,B 0,C 180,E1 -6641.627,E2 -6641.627} C_VEL
LIN {X 0,Y 488.752,Z 379.607,A -85,B 0,C 180,E1 -6644.999,E2 -6644.999} C_VEL
LIN {X 0,Y 488.799,Z 379.601,A -85,B 0,C 180,E1 -6648.387,E2 -6648.387} C_VEL
LIN {X 0,Y 488.809,Z 379.598,A -85,B 0,C 180,E1 -6651.734,E2 -6651.734} C_VEL
LIN {X 0,Y 488.845,Z 379.594,A -85,B 0,C 180,E1 -6654.224,E2 -6654.224} C_VEL
LIN {X 0,Y 488.952,Z 379.579,A -85,B 0,C 180,E1 -6657.529,E2 -6657.529} C_VEL
LIN {X 0,Y 488.959,Z 379.579,A -85,B 0,C 180,E1 -6660,E2 -6660} C_VEL
LIN {X 0,Y 488.952,Z 379.581,A -85,B 0,C 180,E1 -6662.472,E2 -6662.472} C_VEL
LIN {X 0,Y 488.846,Z 379.592,A -85,B 0,C 180,E1 -6665.776,E2 -6665.776} C_VEL
LIN {X 0,Y 488.81,Z 379.6,A -85,B 0,C 180,E1 -6668.267,E2 -6668.267} C_VEL
LIN {X 0,Y 488.799,Z 379.599,A -85,B 0,C 180,E1 -6671.613,E2 -6671.613} C_VEL
LIN {X 0,Y 488.753,Z 379.605,A -85,B 0,C 180,E1 -6675.001,E2 -6675.001} C_VEL
LIN {X 0,Y 488.746,Z 379.607,A -85,B 0,C 180,E1 -6678.443,E2 -6678.443} C_VEL
LIN {X 0,Y 488.7,Z 379.612,A -85,B 0,C 180,E1 -6681.071,E2 -6681.071} C_VEL
LIN {X 0,Y 488.686,Z 379.614,A -85,B 0,C 180,E1 -6683.746,E2 -6683.746} C_VEL
LIN {X 0,Y 488.792,Z 379.601,A -85,B 0,C 180,E1 -6686.946,E2 -6686.946} C_VEL
LIN {X 0,Y 488.703,Z 379.614,A -85,B 0,C 180,E1 -6690.364,E2 -6690.364} C_VEL
LIN {X 0,Y 488.73,Z 379.607,A -85,B 0,C 180,E1 -6693.485,E2 -6693.485} C_VEL
LIN {X 0,Y 488.685,Z 379.614,A -85,B 0,C 180,E1 -6696.357,E2 -6696.357} C_VEL
LIN {X 0,Y 488.744,Z 379.606,A -85,B 0,C 180,E1 -6699.25,E2 -6699.25} C_VEL
LIN {X 0,Y 488.687,Z 379.615,A -85,B 0,C 180,E1 -6702.526,E2 -6702.526} C_VEL
LIN {X 0,Y 488.708,Z 379.609,A -85,B 0,C 180,E1 -6705.2,E2 -6705.2} C_VEL
LIN {X 0,Y 488.706,Z 379.612,A -85,B 0,C 180,E1 -6708.401,E2 -6708.401} C_VEL
LIN {X 0,Y 488.702,Z 379.611,A -85,B 0,C 180,E1 -6710.948,E2 -6710.948} C_VEL
LIN {X 0,Y 488.682,Z 379.615,A -85,B 0,C 180,E1 -6713.869,E2 -6713.869} C_VEL
LIN {X 0,Y 488.738,Z 379.607,A -85,B 0,C 180,E1 -6716.878,E2 -6716.878} C_VEL
LIN {X 0,Y 488.724,Z 379.609,A -85,B 0,C 180,E1 -6719.782,E2 -6719.782} C_VEL
LIN {X 0,Y 488.793,Z 379.598,A -85,B 0,C 180,E1 -6723.057,E2 -6723.057} C_VEL
LIN {X 0,Y 488.744,Z 379.607,A -85,B 0,C 180,E1 -6724.352,E2 -6724.352} C_VEL
LIN {X 0,Y 488.101,Z 379.691,A -85,B 0,C 180,E1 -6725.04,E2 -6725.04} C_VEL
LIN {X 0,Y 485.234,Z 380.05,A -85,B 0,C 180,E1 -6726.156,E2 -6726.156} C_VEL
LIN {X 0,Y 482.788,Z 380.351,A -85,B 0,C 180,E1 -6727.056,E2 -6727.056} C_VEL
LIN {X 0,Y 481.73,Z 380.481,A -85,B 0,C 180,E1 -6727.751,E2 -6727.751} C_VEL
LIN {X 0,Y 481.64,Z 380.49,A -85,B 0,C 180,E1 -6727.987,E2 -6727.987} C_VEL
LIN {X 0,Y 481.707,Z 380.483,A -85,B 0,C 180,E1 -6730.394,E2 -6730.394} C_VEL
LIN {X 0,Y 481.69,Z 380.483,A -85,B 0,C 180,E1 -6733.034,E2 -6733.034} C_VEL
LIN {X 0,Y 481.693,Z 380.486,A -85,B 0,C 180,E1 -6735.639,E2 -6735.639} C_VEL
LIN {X 0,Y 481.755,Z 380.477,A -85,B 0,C 180,E1 -6738.216,E2 -6738.216} C_VEL
LIN {X 0,Y 481.765,Z 380.477,A -85,B 0,C 180,E1 -6741.612,E2 -6741.612} C_VEL
LIN {X 0,Y 481.82,Z 380.469,A -85,B 0,C 180,E1 -6744.14,E2 -6744.14} C_VEL
LIN {X 0,Y 481.723,Z 380.484,A -85,B 0,C 180,E1 -6748.328,E2 -6748.328} C_VEL
LIN {X 0,Y 481.505,Z 380.511,A -85,B 0,C 180,E1 -6750,E2 -6750} C_VEL
LIN {X 0,Y 481.293,Z 384.793,A -85,B 0,C 180,E1 -6754.187,E2 -6754.187} C_VEL
LIN {X 0,Y 481.246,Z 387.545,A -85,B 0,C 180,E1 -6756.753,E2 -6756.753} C_VEL
LIN {X 0,Y 481.06,Z 391.178,A -85,B 0,C 180,E1 -6760.097,E2 -6760.097} C_VEL
LIN {X 0,Y 481.019,Z 393.948,A -85,B 0,C 180,E1 -6762.66,E2 -6762.66} C_VEL
LIN {X 0,Y 481.001,Z 396.909,A -85,B 0,C 180,E1 -6765.346,E2 -6765.346} C_VEL
LIN {X 0,Y 480.968,Z 398.905,A -85,B 0,C 180,E1 -6767.156,E2 -6767.156} C_VEL
LIN {X 0,Y 483.975,Z 412.567,A -85,B 0,C 180,E1 -6767.673,E2 -6767.673} C_VEL
LIN {X 0,Y 483.75,Z 424.889,A -85,B 0,C 180,E1 -6768.201,E2 -6768.201} C_VEL
LIN {X 0,Y 483.32,Z 437.255,A -85,B 0,C 180,E1 -6768.92,E2 -6768.92} C_VEL
LIN {X 0,Y 482.959,Z 448.627,A -85,B 0,C 180,E1 -6769.775,E2 -6769.775} C_VEL
LIN {X 0,Y 482.52,Z 458.074,A -85,B 0,C 180,E1 -6770.653,E2 -6770.653} C_VEL
LIN {X 0,Y 482.164,Z 466.416,A -85,B 0,C 180,E1 -6771.595,E2 -6771.595} C_VEL
LIN {X 0,Y 481.776,Z 474.772,A -85,B 0,C 180,E1 -6772.741,E2 -6772.741} C_VEL
LIN {X 0,Y 481.452,Z 482.854,A -85,B 0,C 180,E1 -6774.125,E2 -6774.125} C_VEL
LIN {X 0,Y 481.206,Z 489.275,A -85,B 0,C 180,E1 -6775.521,E2 -6775.521} C_VEL
LIN {X 0,Y 481.054,Z 494.345,A -85,B 0,C 180,E1 -6776.977,E2 -6776.977} C_VEL
LIN {X 0,Y 480.966,Z 496.789,A -85,B 0,C 180,E1 -6777.878,E2 -6777.878} C_VEL
LIN {X 0,Y 480.883,Z 498.822,A -85,B 0,C 180,E1 -6778.834,E2 -6778.834} C_VEL
LIN {X 0,Y 480.8,Z 500.979,A -85,B 0,C 180,E1 -6780.41,E2 -6780.41} C_VEL
LIN {X 0,Y 480.776,Z 501.766,A -85,B 0,C 180,E1 -6782.021,E2 -6782.021} C_VEL
LIN {X 0,Y 480.788,Z 501.113,A -85,B 0,C 180,E1 -6783.57,E2 -6783.57} C_VEL
LIN {X 0,Y 480.857,Z 499.203,A -85,B 0,C 180,E1 -6785.067,E2 -6785.067} C_VEL
LIN {X 0,Y 481.003,Z 496.092,A -85,B 0,C 180,E1 -6786.523,E2 -6786.523} C_VEL
LIN {X 0,Y 481.128,Z 491.828,A -85,B 0,C 180,E1 -6787.926,E2 -6787.926} C_VEL
LIN {X 0,Y 481.362,Z 486.245,A -85,B 0,C 180,E1 -6789.302,E2 -6789.302} C_VEL
LIN {X 0,Y 481.641,Z 479.297,A -85,B 0,C 180,E1 -6790.643,E2 -6790.643} C_VEL
LIN {X 0,Y 481.992,Z 470.77,A -85,B 0,C 180,E1 -6791.957,E2 -6791.957} C_VEL
LIN {X 0,Y 482.377,Z 461.694,A -85,B 0,C 180,E1 -6793.073,E2 -6793.073} C_VEL
LIN {X 0,Y 482.774,Z 452.097,A -85,B 0,C 180,E1 -6794.036,E2 -6794.036} C_VEL
LIN {X 0,Y 483.203,Z 441.089,A -85,B 0,C 180,E1 -6794.928,E2 -6794.928} C_VEL
LIN {X 0,Y 483.583,Z 430.707,A -85,B 0,C 180,E1 -6795.595,E2 -6795.595} C_VEL
LIN {X 0,Y 483.95,Z 418.287,A -85,B 0,C 180,E1 -6796.205,E2 -6796.205} C_VEL
LIN {X 0,Y 483.877,Z 412.138,A -85,B 0,C 180,E1 -6796.449,E2 -6796.449} C_VEL
LIN {X 0,Y 480.946,Z 399.41,A -85,B 0,C 180,E1 -6796.939,E2 -6796.939} C_VEL
LIN {X 0,Y 480.97,Z 396.136,A -85,B 0,C 180,E1 -6799.989,E2 -6799.989} C_VEL
LIN {X 0,Y 480.994,Z 392.741,A -85,B 0,C 180,E1 -6803.197,E2 -6803.197} C_VEL
LIN {X 0,Y 481.111,Z 390.555,A -85,B 0,C 180,E1 -6805.27,E2 -6805.27} C_VEL
LIN {X 0,Y 481.213,Z 387.412,A -85,B 0,C 180,E1 -6808.28,E2 -6808.28} C_VEL
LIN {X 0,Y 481.246,Z 384.383,A -85,B 0,C 180,E1 -6811.189,E2 -6811.189} C_VEL
LIN {X 0,Y 481.305,Z 381.434,A -85,B 0,C 180,E1 -6814.02,E2 -6814.02} C_VEL
LIN {X 0,Y 481.336,Z 380.533,A -85,B 0,C 180,E1 -6814.948,E2 -6814.948} C_VEL
LIN {X 0,Y 481.618,Z 380.497,A -85,B 0,C 180,E1 -6817.703,E2 -6817.703} C_VEL
LIN {X 0,Y 481.703,Z 380.484,A -85,B 0,C 180,E1 -6820.393,E2 -6820.393} C_VEL
LIN {X 0,Y 481.685,Z 380.486,A -85,B 0,C 180,E1 -6823.034,E2 -6823.034} C_VEL
LIN {X 0,Y 481.683,Z 380.487,A -85,B 0,C 180,E1 -6825.638,E2 -6825.638} C_VEL
LIN {X 0,Y 481.747,Z 380.48,A -85,B 0,C 180,E1 -6828.215,E2 -6828.215} C_VEL
LIN {X 0,Y 481.757,Z 380.478,A -85,B 0,C 180,E1 -6831.611,E2 -6831.611} C_VEL
LIN {X 0,Y 481.81,Z 380.472,A -85,B 0,C 180,E1 -6834.139,E2 -6834.139} C_VEL
LIN {X 0,Y 481.922,Z 380.454,A -85,B 0,C 180,E1 -6837.492,E2 -6837.492} C_VEL
LIN {X 0,Y 481.92,Z 380.456,A -85,B 0,C 180,E1 -6840.836,E2 -6840.836} C_VEL
LIN {X 0,Y 481.921,Z 380.456,A -85,B 0,C 180,E1 -6842.507,E2 -6842.507} C_VEL
LIN {X 0,Y 481.809,Z 380.469,A -85,B 0,C 180,E1 -6845.86,E2 -6845.86} C_VEL
LIN {X 0,Y 481.757,Z 380.475,A -85,B 0,C 180,E1 -6848.388,E2 -6848.388} C_VEL
LIN {X 0,Y 481.746,Z 380.477,A -85,B 0,C 180,E1 -6851.785,E2 -6851.785} C_VEL
LIN {X 0,Y 481.736,Z 380.479,A -85,B 0,C 180,E1 -6855.224,E2 -6855.224} C_VEL
LIN {X 0,Y 481.706,Z 380.482,A -85,B 0,C 180,E1 -6858.722,E2 -6858.722} C_VEL
LIN {X 0,Y 481.64,Z 380.491,A -85,B 0,C 180,E1 -6861.395,E2 -6861.395} C_VEL
LIN {X 0,Y 481.671,Z 380.487,A -85,B 0,C 180,E1 -6864.113,E2 -6864.113} C_VEL
LIN {X 0,Y 481.747,Z 380.48,A -85,B 0,C 180,E1 -6867.141,E2 -6867.141} C_VEL
LIN {X 0,Y 481.674,Z 380.488,A -85,B 0,C 180,E1 -6869.741,E2 -6869.741} C_VEL
LIN {X 0,Y 481.665,Z 380.49,A -85,B 0,C 180,E1 -6872.675,E2 -6872.675} C_VEL
LIN {X 0,Y 481.631,Z 380.496,A -85,B 0,C 180,E1 -6875.71,E2 -6875.71} C_VEL
LIN {X 0,Y 481.717,Z 380.484,A -85,B 0,C 180,E1 -6879.355,E2 -6879.355} C_VEL
LIN {X 0,Y 481.646,Z 380.491,A -85,B 0,C 180,E1 -6882.161,E2 -6882.161} C_VEL
LIN {X 0,Y 481.657,Z 380.491,A -85,B 0,C 180,E1 -6885.543,E2 -6885.543} C_VEL
LIN {X 0,Y 481.665,Z 380.492,A -85,B 0,C 180,E1 -6888.96,E2 -6888.96} C_VEL
LIN {X 0,Y 481.726,Z 380.624,A -85,B 0,C 180,E1 -6889.803,E2 -6889.803} C_VEL
LIN {X 0,Y 483.203,Z 388.679,A -85,B 0,C 180,E1 -6893.393,E2 -6893.393} C_VEL
LIN {X 0,Y 483.199,Z 393.919,A -85,B 0,C 180,E1 -6895.442,E2 -6895.442} C_VEL
LIN {X 0,Y 482.879,Z 400.696,A -85,B 0,C 180,E1 -6897.986,E2 -6897.986} C_VEL
LIN {X 0,Y 482.466,Z 409.826,A -85,B 0,C 180,E1 -6901.269,E2 -6901.269} C_VEL
LIN {X 0,Y 482.196,Z 417.856,A -85,B 0,C 180,E1 -6904.072,E2 -6904.072} C_VEL
LIN {X 0,Y 481.906,Z 427.486,A -85,B 0,C 180,E1 -6907.265,E2 -6907.265} C_VEL
LIN {X 0,Y 481.678,Z 437.194,A -85,B 0,C 180,E1 -6910.392,E2 -6910.392} C_VEL
LIN {X 0,Y 481.434,Z 446.731,A -85,B 0,C 180,E1 -6913.461,E2 -6913.461} C_VEL
LIN {X 0,Y 481.334,Z 451.582,A -85,B 0,C 180,E1 -6915.05,E2 -6915.05} C_VEL
LIN {X 0,Y 483.642,Z 465.098,A -85,B 0,C 180,E1 -6915.456,E2 -6915.456} C_VEL
LIN {X 0,Y 483.933,Z 470.504,A -85,B 0,C 180,E1 -6915.653,E2 -6915.653} C_VEL
LIN {X 0,Y 483.512,Z 483.504,A -85,B 0,C 180,E1 -6916.231,E2 -6916.231} C_VEL
LIN {X 0,Y 483.105,Z 494.678,A -85,B 0,C 180,E1 -6916.894,E2 -6916.894} C_VEL
LIN {X 0,Y 482.758,Z 505.485,A -85,B 0,C 180,E1 -6917.707,E2 -6917.707} C_VEL
LIN {X 0,Y 482.325,Z 515.646,A -85,B 0,C 180,E1 -6918.655,E2 -6918.655} C_VEL
LIN {X 0,Y 481.878,Z 524.786,A -85,B 0,C 180,E1 -6919.708,E2 -6919.708} C_VEL
LIN {X 0,Y 481.531,Z 533.688,A -85,B 0,C 180,E1 -6920.973,E2 -6920.973} C_VEL
LIN {X 0,Y 481.207,Z 540.848,A -85,B 0,C 180,E1 -6922.236,E2 -6922.236} C_VEL
LIN {X 0,Y 481.048,Z 546.357,A -85,B 0,C 180,E1 -6923.448,E2 -6923.448} C_VEL
LIN {X 0,Y 480.998,Z 550.373,A -85,B 0,C 180,E1 -6924.55,E2 -6924.55} C_VEL
LIN {X 0,Y 480.847,Z 553.958,A -85,B 0,C 180,E1 -6925.809,E2 -6925.809} C_VEL
LIN {X 0,Y 480.891,Z 555.807,A -85,B 0,C 180,E1 -6926.649,E2 -6926.649} C_VEL
LIN {X 0,Y 480.79,Z 558.182,A -85,B 0,C 180,E1 -6928.325,E2 -6928.325} C_VEL
LIN {X 0,Y 480.743,Z 559,A -85,B 0,C 180,E1 -6930,E2 -6930} C_VEL
LIN {X 0,Y 480.79,Z 558.184,A -85,B 0,C 180,E1 -6931.675,E2 -6931.675} C_VEL
LIN {X 0,Y 480.891,Z 555.81,A -85,B 0,C 180,E1 -6933.351,E2 -6933.351} C_VEL
LIN {X 0,Y 480.854,Z 552.896,A -85,B 0,C 180,E1 -6934.61,E2 -6934.61} C_VEL
LIN {X 0,Y 481.022,Z 548.949,A -85,B 0,C 180,E1 -6935.87,E2 -6935.87} C_VEL
LIN {X 0,Y 481.116,Z 542.877,A -85,B 0,C 180,E1 -6937.343,E2 -6937.343} C_VEL
LIN {X 0,Y 481.426,Z 536.238,A -85,B 0,C 180,E1 -6938.605,E2 -6938.605} C_VEL
LIN {X 0,Y 481.756,Z 527.995,A -85,B 0,C 180,E1 -6939.87,E2 -6939.87} C_VEL
LIN {X 0,Y 482.115,Z 519.543,A -85,B 0,C 180,E1 -6940.924,E2 -6940.924} C_VEL
LIN {X 0,Y 482.605,Z 509.097,A -85,B 0,C 180,E1 -6941.976,E2 -6941.976} C_VEL
LIN {X 0,Y 482.983,Z 497.276,A -85,B 0,C 180,E1 -6942.931,E2 -6942.931} C_VEL
LIN {X 0,Y 483.409,Z 485.496,A -85,B 0,C 180,E1 -6943.665,E2 -6943.665} C_VEL
LIN {X 0,Y 483.857,Z 473.176,A -85,B 0,C 180,E1 -6944.241,E2 -6944.241} C_VEL
LIN {X 0,Y 483.759,Z 465.936,A -85,B 0,C 180,E1 -6944.513,E2 -6944.513} C_VEL
LIN {X 0,Y 481.603,Z 453.14,A -85,B 0,C 180,E1 -6944.912,E2 -6944.912} C_VEL
LIN {X 0,Y 481.336,Z 451.532,A -85,B 0,C 180,E1 -6944.966,E2 -6944.966} C_VEL
LIN {X 0,Y 481.606,Z 440.801,A -85,B 0,C 180,E1 -6948.461,E2 -6948.461} C_VEL
LIN {X 0,Y 481.824,Z 431.748,A -85,B 0,C 180,E1 -6951.386,E2 -6951.386} C_VEL
LIN {X 0,Y 482.067,Z 422.087,A -85,B 0,C 180,E1 -6954.55,E2 -6954.55} C_VEL
LIN {X 0,Y 482.338,Z 414.197,A -85,B 0,C 180,E1 -6957.275,E2 -6957.275} C_VEL
LIN {X 0,Y 482.738,Z 404.822,A -85,B 0,C 180,E1 -6960.633,E2 -6960.633} C_VEL
LIN {X 0,Y 483.127,Z 396.858,A -85,B 0,C 180,E1 -6963.557,E2 -6963.557} C_VEL
LIN {X 0,Y 483.374,Z 390.35,A -85,B 0,C 180,E1 -6966.074,E2 -6966.074} C_VEL
LIN {X 0,Y 482.593,Z 385.364,A -85,B 0,C 180,E1 -6968.149,E2 -6968.149} C_VEL
LIN {X 0,Y 481.684,Z 380.485,A -85,B 0,C 180,E1 -6970.33,E2 -6970.33} C_VEL
LIN {X 0,Y 481.635,Z 380.493,A -85,B 0,C 180,E1 -6973.299,E2 -6973.299} C_VEL
LIN {X 0,Y 481.653,Z 380.49,A -85,B 0,C 180,E1 -6975.64,E2 -6975.64} C_VEL
LIN {X 0,Y 481.663,Z 380.489,A -85,B 0,C 180,E1 -6978.959,E2 -6978.959} C_VEL
LIN {X 0,Y 481.695,Z 380.485,A -85,B 0,C 180,E1 -6981.143,E2 -6981.143} C_VEL
LIN {X 0,Y 481.662,Z 380.489,A -85,B 0,C 180,E1 -6984.794,E2 -6984.794} C_VEL
LIN {X 0,Y 481.666,Z 380.489,A -85,B 0,C 180,E1 -6987.325,E2 -6987.325} C_VEL
LIN {X 0,Y 481.671,Z 380.486,A -85,B 0,C 180,E1 -6990.258,E2 -6990.258} C_VEL
LIN {X 0,Y 481.744,Z 380.479,A -85,B 0,C 180,E1 -6993.112,E2 -6993.112} C_VEL
LIN {X 0,Y 481.669,Z 380.487,A -85,B 0,C 180,E1 -6995.886,E2 -6995.886} C_VEL
LIN {X 0,Y 481.694,Z 380.485,A -85,B 0,C 180,E1 -6999.027,E2 -6999.027} C_VEL
LIN {X 0,Y 481.699,Z 380.484,A -85,B 0,C 180,E1 -7002.158,E2 -7002.158} C_VEL
LIN {X 0,Y 481.733,Z 380.481,A -85,B 0,C 180,E1 -7004.776,E2 -7004.776} C_VEL
LIN {X 0,Y 481.743,Z 380.478,A -85,B 0,C 180,E1 -7008.215,E2 -7008.215} C_VEL
LIN {X 0,Y 481.755,Z 380.477,A -85,B 0,C 180,E1 -7011.612,E2 -7011.612} C_VEL
LIN {X 0,Y 481.806,Z 380.472,A -85,B 0,C 180,E1 -7014.14,E2 -7014.14} C_VEL
LIN {X 0,Y 481.919,Z 380.455,A -85,B 0,C 180,E1 -7017.493,E2 -7017.493} C_VEL
LIN {X 0,Y 481.93,Z 380.454,A -85,B 0,C 180,E1 -7020,E2 -7020} C_VEL
LIN {X 0,Y 481.919,Z 380.458,A -85,B 0,C 180,E1 -7022.508,E2 -7022.508} C_VEL
LIN {X 0,Y 481.807,Z 380.47,A -85,B 0,C 180,E1 -7025.861,E2 -7025.861} C_VEL
LIN {X 0,Y 481.755,Z 380.479,A -85,B 0,C 180,E1 -7028.389,E2 -7028.389} C_VEL
LIN {X 0,Y 481.744,Z 380.479,A -85,B 0,C 180,E1 -7031.785,E2 -7031.785} C_VEL
LIN {X 0,Y 481.733,Z 380.478,A -85,B 0,C 180,E1 -7035.225,E2 -7035.225} C_VEL
LIN {X 0,Y 481.704,Z 380.484,A -85,B 0,C 180,E1 -7038.722,E2 -7038.722} C_VEL
LIN {X 0,Y 481.639,Z 380.491,A -85,B 0,C 180,E1 -7041.395,E2 -7041.395} C_VEL
LIN {X 0,Y 481.67,Z 380.488,A -85,B 0,C 180,E1 -7044.114,E2 -7044.114} C_VEL
LIN {X 0,Y 481.745,Z 380.478,A -85,B 0,C 180,E1 -7047.141,E2 -7047.141} C_VEL
LIN {X 0,Y 481.672,Z 380.487,A -85,B 0,C 180,E1 -7049.742,E2 -7049.742} C_VEL
LIN {X 0,Y 481.667,Z 380.488,A -85,B 0,C 180,E1 -7052.675,E2 -7052.675} C_VEL
LIN {X 0,Y 481.638,Z 380.491,A -85,B 0,C 180,E1 -7055.71,E2 -7055.71} C_VEL
LIN {X 0,Y 481.715,Z 380.482,A -85,B 0,C 180,E1 -7059.356,E2 -7059.356} C_VEL
LIN {X 0,Y 481.644,Z 380.492,A -85,B 0,C 180,E1 -7062.161,E2 -7062.161} C_VEL
LIN {X 0,Y 481.656,Z 380.488,A -85,B 0,C 180,E1 -7065.544,E2 -7065.544} C_VEL
LIN {X 0,Y 481.654,Z 380.489,A -85,B 0,C 180,E1 -7068.959,E2 -7068.959} C_VEL
LIN {X 0,Y 481.654,Z 380.49,A -85,B 0,C 180,E1 -7071.993,E2 -7071.993} C_VEL
LIN {X 0,Y 481.691,Z 380.484,A -85,B 0,C 180,E1 -7075.319,E2 -7075.319} C_VEL
LIN {X 0,Y 481.645,Z 380.491,A -85,B 0,C 180,E1 -7078.313,E2 -7078.313} C_VEL
LIN {X 0,Y 481.7,Z 380.483,A -85,B 0,C 180,E1 -7081.219,E2 -7081.219} C_VEL
LIN {X 0,Y 481.702,Z 380.484,A -85,B 0,C 180,E1 -7084.044,E2 -7084.044} C_VEL
LIN {X 0,Y 481.676,Z 380.486,A -85,B 0,C 180,E1 -7086.812,E2 -7086.812} C_VEL
LIN {X 0,Y 481.64,Z 380.49,A -85,B 0,C 180,E1 -7087.987,E2 -7087.987} C_VEL
LIN {X 0,Y 480.972,Z 380.574,A -85,B 0,C 180,E1 -7088.685,E2 -7088.685} C_VEL
LIN {X 0,Y 478.145,Z 380.927,A -85,B 0,C 180,E1 -7089.819,E2 -7089.819} C_VEL
LIN {X 0,Y 475.76,Z 381.224,A -85,B 0,C 180,E1 -7090.733,E2 -7090.733} C_VEL
LIN {X 0,Y 474.739,Z 381.352,A -85,B 0,C 180,E1 -7091.439,E2 -7091.439} C_VEL
LIN {X 0,Y 474.657,Z 381.361,A -85,B 0,C 180,E1 -7091.678,E2 -7091.678} C_VEL
LIN {X 0,Y 474.703,Z 381.355,A -85,B 0,C 180,E1 -7094.545,E2 -7094.545} C_VEL
LIN {X 0,Y 474.708,Z 381.356,A -85,B 0,C 180,E1 -7098.038,E2 -7098.038} C_VEL
LIN {X 0,Y 474.73,Z 381.354,A -85,B 0,C 180,E1 -7101.487,E2 -7101.487} C_VEL
LIN {X 0,Y 474.783,Z 381.346,A -85,B 0,C 180,E1 -7104.053,E2 -7104.053} C_VEL
LIN {X 0,Y 474.696,Z 381.359,A -85,B 0,C 180,E1 -7108.303,E2 -7108.303} C_VEL
LIN {X 0,Y 474.479,Z 381.386,A -85,B 0,C 180,E1 -7110,E2 -7110} C_VEL
LIN {X 0,Y 474.066,Z 383.796,A -85,B 0,C 180,E1 -7112.549,E2 -7112.549} C_VEL
LIN {X 0,Y 474.196,Z 386.494,A -85,B 0,C 180,E1 -7115.102,E2 -7115.102} C_VEL
LIN {X 0,Y 474.113,Z 389.232,A -85,B 0,C 180,E1 -7117.667,E2 -7117.667} C_VEL
LIN {X 0,Y 474.046,Z 392.939,A -85,B 0,C 180,E1 -7121.112,E2 -7121.112} C_VEL
LIN {X 0,Y 473.959,Z 396.7,A -85,B 0,C 180,E1 -7124.601,E2 -7124.601} C_VEL
LIN {X 0,Y 473.874,Z 399.333,A -85,B 0,C 180,E1 -7126.949,E2 -7126.949} C_VEL
LIN {X 0,Y 477.058,Z 413.097,A -85,B 0,C 180,E1 -7127.467,E2 -7127.467} C_VEL
LIN {X 0,Y 476.906,Z 424.699,A -85,B 0,C 180,E1 -7127.972,E2 -7127.972} C_VEL
LIN {X 0,Y 476.493,Z 435.74,A -85,B 0,C 180,E1 -7128.6,E2 -7128.6} C_VEL
LIN {X 0,Y 476.058,Z 447.316,A -85,B 0,C 180,E1 -7129.452,E2 -7129.452} C_VEL
LIN {X 0,Y 475.585,Z 457.949,A -85,B 0,C 180,E1 -7130.433,E2 -7130.433} C_VEL
LIN {X 0,Y 475.149,Z 467.772,A -85,B 0,C 180,E1 -7131.564,E2 -7131.564} C_VEL
LIN {X 0,Y 474.685,Z 476.486,A -85,B 0,C 180,E1 -7132.81,E2 -7132.81} C_VEL
LIN {X 0,Y 474.418,Z 483.436,A -85,B 0,C 180,E1 -7134.04,E2 -7134.04} C_VEL
LIN {X 0,Y 474.153,Z 489.823,A -85,B 0,C 180,E1 -7135.457,E2 -7135.457} C_VEL
LIN {X 0,Y 474.005,Z 494.436,A -85,B 0,C 180,E1 -7136.787,E2 -7136.787} C_VEL
LIN {X 0,Y 473.835,Z 498.362,A -85,B 0,C 180,E1 -7138.335,E2 -7138.335} C_VEL
LIN {X 0,Y 473.768,Z 500.133,A -85,B 0,C 180,E1 -7139.309,E2 -7139.309} C_VEL
LIN {X 0,Y 473.728,Z 501.64,A -85,B 0,C 180,E1 -7140.631,E2 -7140.631} C_VEL
LIN {X 0,Y 473.692,Z 502.164,A -85,B 0,C 180,E1 -7142.284,E2 -7142.284} C_VEL
LIN {X 0,Y 473.706,Z 501.345,A -85,B 0,C 180,E1 -7143.816,E2 -7143.816} C_VEL
LIN {X 0,Y 473.814,Z 499.254,A -85,B 0,C 180,E1 -7145.343,E2 -7145.343} C_VEL
LIN {X 0,Y 473.974,Z 495.991,A -85,B 0,C 180,E1 -7146.802,E2 -7146.802} C_VEL
LIN {X 0,Y 474.107,Z 491.523,A -85,B 0,C 180,E1 -7148.218,E2 -7148.218} C_VEL
LIN {X 0,Y 474.34,Z 485.781,A -85,B 0,C 180,E1 -7149.605,E2 -7149.605} C_VEL
LIN {X 0,Y 474.672,Z 478.637,A -85,B 0,C 180,E1 -7150.965,E2 -7150.965} C_VEL
LIN {X 0,Y 474.994,Z 471.779,A -85,B 0,C 180,E1 -7152.022,E2 -7152.022} C_VEL
LIN {X 0,Y 475.399,Z 463.127,A -85,B 0,C 180,E1 -7153.126,E2 -7153.126} C_VEL
LIN {X 0,Y 475.79,Z 453.617,A -85,B 0,C 180,E1 -7154.114,E2 -7154.114} C_VEL
LIN {X 0,Y 476.203,Z 443.714,A -85,B 0,C 180,E1 -7154.952,E2 -7154.952} C_VEL
LIN {X 0,Y 476.646,Z 432.251,A -85,B 0,C 180,E1 -7155.728,E2 -7155.728} C_VEL
LIN {X 0,Y 477.062,Z 419.965,A -85,B 0,C 180,E1 -7156.361,E2 -7156.361} C_VEL
LIN {X 0,Y 477.003,Z 413.155,A -85,B 0,C 180,E1 -7156.639,E2 -7156.639} C_VEL
LIN {X 0,Y 473.892,Z 399.859,A -85,B 0,C 180,E1 -7157.163,E2 -7157.163} C_VEL
LIN {X 0,Y 473.909,Z 396.341,A -85,B 0,C 180,E1 -7160.456,E2 -7160.456} C_VEL
LIN {X 0,Y 473.952,Z 393.033,A -85,B 0,C 180,E1 -7163.62,E2 -7163.62} C_VEL
LIN {X 0,Y 474.09,Z 389.808,A -85,B 0,C 180,E1 -7166.736,E2 -7166.736} C_VEL
LIN {X 0,Y 474.156,Z 386.679,A -85,B 0,C 180,E1 -7169.738,E2 -7169.738} C_VEL
LIN {X 0,Y 474.19,Z 383.536,A -85,B 0,C 180,E1 -7172.779,E2 -7172.779} C_VEL
LIN {X 0,Y 474.283,Z 381.576,A -85,B 0,C 180,E1 -7174.675,E2 -7174.675} C_VEL
LIN {X 0,Y 474.552,Z 381.379,A -85,B 0,C 180,E1 -7177.353,E2 -7177.353} C_VEL
LIN {X 0,Y 474.652,Z 381.363,A -85,B 0,C 180,E1 -7180.089,E2 -7180.089} C_VEL
LIN {X 0,Y 474.645,Z 381.362,A -85,B 0,C 180,E1 -7182.774,E2 -7182.774} C_VEL
LIN {X 0,Y 474.642,Z 381.363,A -85,B 0,C 180,E1 -7185.421,E2 -7185.421} C_VEL
LIN {X 0,Y 474.7,Z 381.357,A -85,B 0,C 180,E1 -7188.037,E2 -7188.037} C_VEL
LIN {X 0,Y 474.723,Z 381.353,A -85,B 0,C 180,E1 -7191.486,E2 -7191.486} C_VEL
LIN {X 0,Y 474.773,Z 381.348,A -85,B 0,C 180,E1 -7194.052,E2 -7194.052} C_VEL
LIN {X 0,Y 474.889,Z 381.33,A -85,B 0,C 180,E1 -7197.455,E2 -7197.455} C_VEL
LIN {X 0,Y 474.871,Z 381.334,A -85,B 0,C 180,E1 -7200.848,E2 -7200.848} C_VEL
LIN {X 0,Y 474.887,Z 381.332,A -85,B 0,C 180,E1 -7202.545,E2 -7202.545} C_VEL
LIN {X 0,Y 474.772,Z 381.346,A -85,B 0,C 180,E1 -7205.948,E2 -7205.948} C_VEL
LIN {X 0,Y 474.722,Z 381.352,A -85,B 0,C 180,E1 -7208.514,E2 -7208.514} C_VEL
LIN {X 0,Y 474.699,Z 381.355,A -85,B 0,C 180,E1 -7211.963,E2 -7211.963} C_VEL
LIN {X 0,Y 474.694,Z 381.355,A -85,B 0,C 180,E1 -7215.456,E2 -7215.456} C_VEL
LIN {X 0,Y 474.659,Z 381.358,A -85,B 0,C 180,E1 -7219.01,E2 -7219.01} C_VEL
LIN {X 0,Y 474.583,Z 381.37,A -85,B 0,C 180,E1 -7221.729,E2 -7221.729} C_VEL
LIN {X 0,Y 474.654,Z 381.364,A -85,B 0,C 180,E1 -7224.493,E2 -7224.493} C_VEL
LIN {X 0,Y 474.694,Z 381.357,A -85,B 0,C 180,E1 -7227.339,E2 -7227.339} C_VEL
LIN {X 0,Y 474.599,Z 381.369,A -85,B 0,C 180,E1 -7230.81,E2 -7230.81} C_VEL
LIN {X 0,Y 474.62,Z 381.368,A -85,B 0,C 180,E1 -7233.222,E2 -7233.222} C_VEL
LIN {X 0,Y 474.584,Z 381.373,A -85,B 0,C 180,E1 -7236.324,E2 -7236.324} C_VEL
LIN {X 0,Y 474.652,Z 381.363,A -85,B 0,C 180,E1 -7239.652,E2 -7239.652} C_VEL
LIN {X 0,Y 474.612,Z 381.367,A -85,B 0,C 180,E1 -7242.935,E2 -7242.935} C_VEL
LIN {X 0,Y 474.607,Z 381.369,A -85,B 0,C 180,E1 -7245.896,E2 -7245.896} C_VEL
LIN {X 0,Y 474.639,Z 381.367,A -85,B 0,C 180,E1 -7249.04,E2 -7249.04} C_VEL
LIN {X 0,Y 474.685,Z 381.478,A -85,B 0,C 180,E1 -7249.478,E2 -7249.478} C_VEL
LIN {X 0,Y 476.022,Z 388.948,A -85,B 0,C 180,E1 -7252.869,E2 -7252.869} C_VEL
LIN {X 0,Y 476.334,Z 392.138,A -85,B 0,C 180,E1 -7254.242,E2 -7254.242} C_VEL
LIN {X 0,Y 475.965,Z 400.07,A -85,B 0,C 180,E1 -7257.315,E2 -7257.315} C_VEL
LIN {X 0,Y 475.53,Z 408.197,A -85,B 0,C 180,E1 -7260.315,E2 -7260.315} C_VEL
LIN {X 0,Y 475.247,Z 416.263,A -85,B 0,C 180,E1 -7263.19,E2 -7263.19} C_VEL
LIN {X 0,Y 474.91,Z 425.729,A -85,B 0,C 180,E1 -7266.45,E2 -7266.45} C_VEL
LIN {X 0,Y 474.686,Z 435.456,A -85,B 0,C 180,E1 -7269.639,E2 -7269.639} C_VEL
LIN {X 0,Y 474.465,Z 443.733,A -85,B 0,C 180,E1 -7272.323,E2 -7272.323} C_VEL
LIN {X 0,Y 474.292,Z 451.601,A -85,B 0,C 180,E1 -7274.827,E2 -7274.827} C_VEL
LIN {X 0,Y 476.608,Z 465.098,A -85,B 0,C 180,E1 -7275.237,E2 -7275.237} C_VEL
LIN {X 0,Y 477.044,Z 470.504,A -85,B 0,C 180,E1 -7275.441,E2 -7275.441} C_VEL
LIN {X 0,Y 476.63,Z 483.504,A -85,B 0,C 180,E1 -7276.028,E2 -7276.028} C_VEL
LIN {X 0,Y 476.197,Z 494.677,A -85,B 0,C 180,E1 -7276.7,E2 -7276.7} C_VEL
LIN {X 0,Y 475.795,Z 505.564,A -85,B 0,C 180,E1 -7277.531,E2 -7277.531} C_VEL
LIN {X 0,Y 475.366,Z 515.646,A -85,B 0,C 180,E1 -7278.487,E2 -7278.487} C_VEL
LIN {X 0,Y 474.88,Z 524.785,A -85,B 0,C 180,E1 -7279.555,E2 -7279.555} C_VEL
LIN {X 0,Y 474.482,Z 533.687,A -85,B 0,C 180,E1 -7280.838,E2 -7280.838} C_VEL
LIN {X 0,Y 474.152,Z 540.848,A -85,B 0,C 180,E1 -7282.12,E2 -7282.12} C_VEL
LIN {X 0,Y 473.972,Z 546.738,A -85,B 0,C 180,E1 -7283.449,E2 -7283.449} C_VEL
LIN {X 0,Y 473.845,Z 551.676,A -85,B 0,C 180,E1 -7284.894,E2 -7284.894} C_VEL
LIN {X 0,Y 473.752,Z 553.957,A -85,B 0,C 180,E1 -7285.746,E2 -7285.746} C_VEL
LIN {X 0,Y 473.799,Z 555.806,A -85,B 0,C 180,E1 -7286.598,E2 -7286.598} C_VEL
LIN {X 0,Y 473.695,Z 558.182,A -85,B 0,C 180,E1 -7288.299,E2 -7288.299} C_VEL
LIN {X 0,Y 473.688,Z 558.785,A -85,B 0,C 180,E1 -7289.15,E2 -7289.15} C_VEL
LIN {X 0,Y 473.669,Z 559,A -85,B 0,C 180,E1 -7290,E2 -7290} C_VEL
LIN {X 0,Y 473.688,Z 558.786,A -85,B 0,C 180,E1 -7290.85,E2 -7290.85} C_VEL
LIN {X 0,Y 473.724,Z 557.196,A -85,B 0,C 180,E1 -7292.551,E2 -7292.551} C_VEL
LIN {X 0,Y 473.799,Z 555.81,A -85,B 0,C 180,E1 -7293.401,E2 -7293.401} C_VEL
LIN {X 0,Y 473.775,Z 552.896,A -85,B 0,C 180,E1 -7294.679,E2 -7294.679} C_VEL
LIN {X 0,Y 473.941,Z 548.949,A -85,B 0,C 180,E1 -7295.958,E2 -7295.958} C_VEL
LIN {X 0,Y 474.049,Z 542.877,A -85,B 0,C 180,E1 -7297.453,E2 -7297.453} C_VEL
LIN {X 0,Y 474.377,Z 536.237,A -85,B 0,C 180,E1 -7298.734,E2 -7298.734} C_VEL
LIN {X 0,Y 474.751,Z 527.995,A -85,B 0,C 180,E1 -7300.017,E2 -7300.017} C_VEL
LIN {X 0,Y 475.132,Z 519.544,A -85,B 0,C 180,E1 -7301.086,E2 -7301.086} C_VEL
LIN {X 0,Y 475.634,Z 509.096,A -85,B 0,C 180,E1 -7302.155,E2 -7302.155} C_VEL
LIN {X 0,Y 476.037,Z 497.916,A -85,B 0,C 180,E1 -7303.075,E2 -7303.075} C_VEL
LIN {X 0,Y 476.452,Z 487.412,A -85,B 0,C 180,E1 -7303.759,E2 -7303.759} C_VEL
LIN {X 0,Y 476.894,Z 475.776,A -85,B 0,C 180,E1 -7304.345,E2 -7304.345} C_VEL
LIN {X 0,Y 476.929,Z 467.079,A -85,B 0,C 180,E1 -7304.684,E2 -7304.684} C_VEL
LIN {X 0,Y 474.753,Z 454.192,A -85,B 0,C 180,E1 -7305.111,E2 -7305.111} C_VEL
LIN {X 0,Y 474.271,Z 451.46,A -85,B 0,C 180,E1 -7305.194,E2 -7305.194} C_VEL
LIN {X 0,Y 474.548,Z 440.995,A -85,B 0,C 180,E1 -7308.588,E2 -7308.588} C_VEL
LIN {X 0,Y 474.811,Z 431.456,A -85,B 0,C 180,E1 -7311.718,E2 -7311.718} C_VEL
LIN {X 0,Y 475.05,Z 421.788,A -85,B 0,C 180,E1 -7314.937,E2 -7314.937} C_VEL
LIN {X 0,Y 475.375,Z 413.715,A -85,B 0,C 180,E1 -7317.812,E2 -7317.812} C_VEL
LIN {X 0,Y 475.778,Z 404.618,A -85,B 0,C 180,E1 -7321.131,E2 -7321.131} C_VEL
LIN {X 0,Y 476.221,Z 396.32,A -85,B 0,C 180,E1 -7324.265,E2 -7324.265} C_VEL
LIN {X 0,Y 476.384,Z 391.513,A -85,B 0,C 180,E1 -7326.164,E2 -7326.164} C_VEL
LIN {X 0,Y 475.527,Z 386.176,A -85,B 0,C 180,E1 -7328.435,E2 -7328.435} C_VEL
LIN {X 0,Y 474.613,Z 381.367,A -85,B 0,C 180,E1 -7330.657,E2 -7330.657} C_VEL
LIN {X 0,Y 474.597,Z 381.37,A -85,B 0,C 180,E1 -7333.48,E2 -7333.48} C_VEL
LIN {X 0,Y 474.596,Z 381.37,A -85,B 0,C 180,E1 -7336.518,E2 -7336.518} C_VEL
LIN {X 0,Y 474.632,Z 381.366,A -85,B 0,C 180,E1 -7339.344,E2 -7339.344} C_VEL
LIN {X 0,Y 474.612,Z 381.368,A -85,B 0,C 180,E1 -7341.702,E2 -7341.702} C_VEL
LIN {X 0,Y 474.624,Z 381.366,A -85,B 0,C 180,E1 -7344.726,E2 -7344.726} C_VEL
LIN {X 0,Y 474.63,Z 381.363,A -85,B 0,C 180,E1 -7347.787,E2 -7347.787} C_VEL
LIN {X 0,Y 474.616,Z 381.367,A -85,B 0,C 180,E1 -7350.884,E2 -7350.884} C_VEL
LIN {X 0,Y 474.659,Z 381.361,A -85,B 0,C 180,E1 -7353.628,E2 -7353.628} C_VEL
LIN {X 0,Y 474.627,Z 381.365,A -85,B 0,C 180,E1 -7356.641,E2 -7356.641} C_VEL
LIN {X 0,Y 474.648,Z 381.361,A -85,B 0,C 180,E1 -7360.089,E2 -7360.089} C_VEL
LIN {X 0,Y 474.642,Z 381.365,A -85,B 0,C 180,E1 -7362.774,E2 -7362.774} C_VEL
LIN {X 0,Y 474.638,Z 381.362,A -85,B 0,C 180,E1 -7365.421,E2 -7365.421} C_VEL
LIN {X 0,Y 474.696,Z 381.355,A -85,B 0,C 180,E1 -7368.037,E2 -7368.037} C_VEL
LIN {X 0,Y 474.72,Z 381.353,A -85,B 0,C 180,E1 -7371.486,E2 -7371.486} C_VEL
LIN {X 0,Y 474.769,Z 381.348,A -85,B 0,C 180,E1 -7374.052,E2 -7374.052} C_VEL
LIN {X 0,Y 474.885,Z 381.331,A -85,B 0,C 180,E1 -7377.455,E2 -7377.455} C_VEL
LIN {X 0,Y 474.868,Z 381.335,A -85,B 0,C 180,E1 -7380.848,E2 -7380.848} C_VEL
LIN {X 0,Y 474.886,Z 381.334,A -85,B 0,C 180,E1 -7382.545,E2 -7382.545} C_VEL
LIN {X 0,Y 474.77,Z 381.346,A -85,B 0,C 180,E1 -7385.948,E2 -7385.948} C_VEL
LIN {X 0,Y 474.72,Z 381.354,A -85,B 0,C 180,E1 -7388.514,E2 -7388.514} C_VEL
LIN {X 0,Y 474.696,Z 381.357,A -85,B 0,C 180,E1 -7391.963,E2 -7391.963} C_VEL
LIN {X 0,Y 474.691,Z 381.355,A -85,B 0,C 180,E1 -7395.456,E2 -7395.456} C_VEL
LIN {X 0,Y 474.657,Z 381.362,A -85,B 0,C 180,E1 -7399.011,E2 -7399.011} C_VEL
LIN {X 0,Y 474.582,Z 381.371,A -85,B 0,C 180,E1 -7401.729,E2 -7401.729} C_VEL
LIN {X 0,Y 474.651,Z 381.363,A -85,B 0,C 180,E1 -7404.493,E2 -7404.493} C_VEL
LIN {X 0,Y 474.692,Z 381.356,A -85,B 0,C 180,E1 -7407.339,E2 -7407.339} C_VEL
LIN {X 0,Y 474.598,Z 381.368,A -85,B 0,C 180,E1 -7410.811,E2 -7410.811} C_VEL
LIN {X 0,Y 474.633,Z 381.365,A -85,B 0,C 180,E1 -7413.985,E2 -7413.985} C_VEL
LIN {X 0,Y 474.571,Z 381.372,A -85,B 0,C 180,E1 -7416.901,E2 -7416.901} C_VEL
LIN {X 0,Y 474.65,Z 381.362,A -85,B 0,C 180,E1 -7419.653,E2 -7419.653} C_VEL
LIN {X 0,Y 474.61,Z 381.365,A -85,B 0,C 180,E1 -7422.935,E2 -7422.935} C_VEL
LIN {X 0,Y 474.606,Z 381.369,A -85,B 0,C 180,E1 -7425.896,E2 -7425.896} C_VEL
LIN {X 0,Y 474.625,Z 381.364,A -85,B 0,C 180,E1 -7429.042,E2 -7429.042} C_VEL
LIN {X 0,Y 474.609,Z 381.368,A -85,B 0,C 180,E1 -7431.705,E2 -7431.705} C_VEL
LIN {X 0,Y 474.628,Z 381.364,A -85,B 0,C 180,E1 -7434.727,E2 -7434.727} C_VEL
LIN {X 0,Y 474.636,Z 381.364,A -85,B 0,C 180,E1 -7437.789,E2 -7437.789} C_VEL
LIN {X 0,Y 474.624,Z 381.364,A -85,B 0,C 180,E1 -7440.885,E2 -7440.885} C_VEL
LIN {X 0,Y 474.662,Z 381.362,A -85,B 0,C 180,E1 -7443.629,E2 -7443.629} C_VEL
LIN {X 0,Y 474.638,Z 381.364,A -85,B 0,C 180,E1 -7446.642,E2 -7446.642} C_VEL
LIN {X 0,Y 474.657,Z 381.363,A -85,B 0,C 180,E1 -7450.09,E2 -7450.09} C_VEL
LIN {X 0,Y 474.657,Z 381.361,A -85,B 0,C 180,E1 -7451.678,E2 -7451.678} C_VEL
LIN {X 0,Y 473.993,Z 381.445,A -85,B 0,C 180,E1 -7452.387,E2 -7452.387} C_VEL
LIN {X 0,Y 471.143,Z 381.801,A -85,B 0,C 180,E1 -7453.539,E2 -7453.539} C_VEL
LIN {X 0,Y 468.727,Z 382.1,A -85,B 0,C 180,E1 -7454.467,E2 -7454.467} C_VEL
LIN {X 0,Y 467.687,Z 382.229,A -85,B 0,C 180,E1 -7455.184,E2 -7455.184} C_VEL
LIN {X 0,Y 467.6,Z 382.238,A -85,B 0,C 180,E1 -7455.427,E2 -7455.427} C_VEL
LIN {X 0,Y 467.655,Z 382.232,A -85,B 0,C 180,E1 -7458.734,E2 -7458.734} C_VEL
LIN {X 0,Y 467.753,Z 382.222,A -85,B 0,C 180,E1 -7462.229,E2 -7462.229} C_VEL
LIN {X 0,Y 467.728,Z 382.223,A -85,B 0,C 180,E1 -7464.828,E2 -7464.828} C_VEL
LIN {X 0,Y 467.669,Z 382.234,A -85,B 0,C 180,E1 -7468.278,E2 -7468.278} C_VEL
LIN {X 0,Y 467.452,Z 382.261,A -85,B 0,C 180,E1 -7470,E2 -7470} C_VEL
LIN {X 0,Y 467.202,Z 382.752,A -85,B 0,C 180,E1 -7470.862,E2 -7470.862} C_VEL
LIN {X 0,Y 467.167,Z 386.359,A -85,B 0,C 180,E1 -7474.314,E2 -7474.314} C_VEL
LIN {X 0,Y 467.117,Z 389.108,A -85,B 0,C 180,E1 -7476.913,E2 -7476.913} C_VEL
LIN {X 0,Y 466.94,Z 392.86,A -85,B 0,C 180,E1 -7480.406,E2 -7480.406} C_VEL
LIN {X 0,Y 466.892,Z 395.694,A -85,B 0,C 180,E1 -7483.049,E2 -7483.049} C_VEL
LIN {X 0,Y 466.844,Z 398.629,A -85,B 0,C 180,E1 -7485.722,E2 -7485.722} C_VEL
LIN {X 0,Y 466.796,Z 399.708,A -85,B 0,C 180,E1 -7486.707,E2 -7486.707} C_VEL
LIN {X 0,Y 470.185,Z 414.316,A -85,B 0,C 180,E1 -7487.282,E2 -7487.282} C_VEL
LIN {X 0,Y 469.953,Z 426.805,A -85,B 0,C 180,E1 -7487.853,E2 -7487.853} C_VEL
LIN {X 0,Y 469.536,Z 438.243,A -85,B 0,C 180,E1 -7488.546,E2 -7488.546} C_VEL
LIN {X 0,Y 469.094,Z 449.875,A -85,B 0,C 180,E1 -7489.449,E2 -7489.449} C_VEL
LIN {X 0,Y 468.588,Z 459.75,A -85,B 0,C 180,E1 -7490.408,E2 -7490.408} C_VEL
LIN {X 0,Y 468.155,Z 468.473,A -85,B 0,C 180,E1 -7491.447,E2 -7491.447} C_VEL
LIN {X 0,Y 467.67,Z 477.472,A -85,B 0,C 180,E1 -7492.765,E2 -7492.765} C_VEL
LIN {X 0,Y 467.388,Z 484.017,A -85,B 0,C 180,E1 -7493.953,E2 -7493.953} C_VEL
LIN {X 0,Y 467.136,Z 489.564,A -85,B 0,C 180,E1 -7495.19,E2 -7495.19} C_VEL
LIN {X 0,Y 466.973,Z 493.76,A -85,B 0,C 180,E1 -7496.358,E2 -7496.358} C_VEL
LIN {X 0,Y 466.817,Z 497.806,A -85,B 0,C 180,E1 -7497.821,E2 -7497.821} C_VEL
LIN {X 0,Y 466.71,Z 500.355,A -85,B 0,C 180,E1 -7499.143,E2 -7499.143} C_VEL
LIN {X 0,Y 466.652,Z 502.224,A -85,B 0,C 180,E1 -7500.857,E2 -7500.857} C_VEL
LIN {X 0,Y 466.603,Z 502.564,A -85,B 0,C 180,E1 -7502.49,E2 -7502.49} C_VEL
LIN {X 0,Y 466.651,Z 501.573,A -85,B 0,C 180,E1 -7504.072,E2 -7504.072} C_VEL
LIN {X 0,Y 466.767,Z 499.304,A -85,B 0,C 180,E1 -7505.603,E2 -7505.603} C_VEL
LIN {X 0,Y 466.916,Z 495.844,A -85,B 0,C 180,E1 -7507.083,E2 -7507.083} C_VEL
LIN {X 0,Y 467.122,Z 491.186,A -85,B 0,C 180,E1 -7508.523,E2 -7508.523} C_VEL
LIN {X 0,Y 467.353,Z 485.3,A -85,B 0,C 180,E1 -7509.92,E2 -7509.92} C_VEL
LIN {X 0,Y 467.717,Z 477.905,A -85,B 0,C 180,E1 -7511.296,E2 -7511.296} C_VEL
LIN {X 0,Y 468.137,Z 469.855,A -85,B 0,C 180,E1 -7512.498,E2 -7512.498} C_VEL
LIN {X 0,Y 468.596,Z 460.626,A -85,B 0,C 180,E1 -7513.622,E2 -7513.622} C_VEL
LIN {X 0,Y 469.074,Z 450.198,A -85,B 0,C 180,E1 -7514.647,E2 -7514.647} C_VEL
LIN {X 0,Y 469.515,Z 438.651,A -85,B 0,C 180,E1 -7515.547,E2 -7515.547} C_VEL
LIN {X 0,Y 469.98,Z 427.267,A -85,B 0,C 180,E1 -7516.238,E2 -7516.238} C_VEL
LIN {X 0,Y 470.295,Z 415.151,A -85,B 0,C 180,E1 -7516.794,E2 -7516.794} C_VEL
LIN {X 0,Y 467.336,Z 402.632,A -85,B 0,C 180,E1 -7517.301,E2 -7517.301} C_VEL
LIN {X 0,Y 466.819,Z 400.327,A -85,B 0,C 180,E1 -7517.384,E2 -7517.384} C_VEL
LIN {X 0,Y 466.832,Z 397.393,A -85,B 0,C 180,E1 -7520.155,E2 -7520.155} C_VEL
LIN {X 0,Y 466.902,Z 394.449,A -85,B 0,C 180,E1 -7522.979,E2 -7522.979} C_VEL
LIN {X 0,Y 467.022,Z 391.158,A -85,B 0,C 180,E1 -7526.165,E2 -7526.165} C_VEL
LIN {X 0,Y 467.123,Z 387.982,A -85,B 0,C 180,E1 -7529.233,E2 -7529.233} C_VEL
LIN {X 0,Y 467.137,Z 384.57,A -85,B 0,C 180,E1 -7532.577,E2 -7532.577} C_VEL
LIN {X 0,Y 467.219,Z 382.603,A -85,B 0,C 180,E1 -7534.491,E2 -7534.491} C_VEL
LIN {X 0,Y 467.371,Z 382.272,A -85,B 0,C 180,E1 -7536.045,E2 -7536.045} C_VEL
LIN {X 0,Y 467.577,Z 382.245,A -85,B 0,C 180,E1 -7538.854,E2 -7538.854} C_VEL
LIN {X 0,Y 467.627,Z 382.237,A -85,B 0,C 180,E1 -7541.602,E2 -7541.602} C_VEL
LIN {X 0,Y 467.633,Z 382.236,A -85,B 0,C 180,E1 -7544.305,E2 -7544.305} C_VEL
LIN {X 0,Y 467.651,Z 382.234,A -85,B 0,C 180,E1 -7547.854,E2 -7547.854} C_VEL
LIN {X 0,Y 467.676,Z 382.23,A -85,B 0,C 180,E1 -7551.357,E2 -7551.357} C_VEL
LIN {X 0,Y 467.738,Z 382.224,A -85,B 0,C 180,E1 -7553.962,E2 -7553.962} C_VEL
LIN {X 0,Y 467.854,Z 382.206,A -85,B 0,C 180,E1 -7557.417,E2 -7557.417} C_VEL
LIN {X 0,Y 467.875,Z 382.204,A -85,B 0,C 180,E1 -7560,E2 -7560} C_VEL
LIN {X 0,Y 467.853,Z 382.208,A -85,B 0,C 180,E1 -7562.583,E2 -7562.583} C_VEL
LIN {X 0,Y 467.736,Z 382.223,A -85,B 0,C 180,E1 -7566.037,E2 -7566.037} C_VEL
LIN {X 0,Y 467.676,Z 382.23,A -85,B 0,C 180,E1 -7568.643,E2 -7568.643} C_VEL
LIN {X 0,Y 467.651,Z 382.234,A -85,B 0,C 180,E1 -7572.146,E2 -7572.146} C_VEL
LIN {X 0,Y 467.633,Z 382.235,A -85,B 0,C 180,E1 -7575.695,E2 -7575.695} C_VEL
LIN {X 0,Y 467.611,Z 382.237,A -85,B 0,C 180,E1 -7578.765,E2 -7578.765} C_VEL
LIN {X 0,Y 467.575,Z 382.243,A -85,B 0,C 180,E1 -7581.268,E2 -7581.268} C_VEL
LIN {X 0,Y 467.568,Z 382.244,A -85,B 0,C 180,E1 -7583.944,E2 -7583.944} C_VEL
LIN {X 0,Y 467.623,Z 382.237,A -85,B 0,C 180,E1 -7586.8,E2 -7586.8} C_VEL
LIN {X 0,Y 467.549,Z 382.248,A -85,B 0,C 180,E1 -7589.739,E2 -7589.739} C_VEL
LIN {X 0,Y 467.574,Z 382.246,A -85,B 0,C 180,E1 -7592.759,E2 -7592.759} C_VEL
LIN {X 0,Y 467.549,Z 382.249,A -85,B 0,C 180,E1 -7595.89,E2 -7595.89} C_VEL
LIN {X 0,Y 467.615,Z 382.241,A -85,B 0,C 180,E1 -7599.142,E2 -7599.142} C_VEL
LIN {X 0,Y 467.584,Z 382.244,A -85,B 0,C 180,E1 -7602.567,E2 -7602.567} C_VEL
LIN {X 0,Y 467.568,Z 382.247,A -85,B 0,C 180,E1 -7605.054,E2 -7605.054} C_VEL
LIN {X 0,Y 467.587,Z 382.247,A -85,B 0,C 180,E1 -7607.44,E2 -7607.44} C_VEL
LIN {X 0,Y 467.623,Z 382.4,A -85,B 0,C 180,E1 -7609.174,E2 -7609.174} C_VEL
LIN {X 0,Y 468.963,Z 389.733,A -85,B 0,C 180,E1 -7612.587,E2 -7612.587} C_VEL
LIN {X 0,Y 469.371,Z 393.604,A -85,B 0,C 180,E1 -7614.271,E2 -7614.271} C_VEL
LIN {X 0,Y 468.949,Z 401.403,A -85,B 0,C 180,E1 -7617.349,E2 -7617.349} C_VEL
LIN {X 0,Y 468.473,Z 409.693,A -85,B 0,C 180,E1 -7620.472,E2 -7620.472} C_VEL
LIN {X 0,Y 468.203,Z 417.341,A -85,B 0,C 180,E1 -7623.236,E2 -7623.236} C_VEL
LIN {X 0,Y 467.859,Z 426.319,A -85,B 0,C 180,E1 -7626.394,E2 -7626.394} C_VEL
LIN {X 0,Y 467.583,Z 436.481,A -85,B 0,C 180,E1 -7629.776,E2 -7629.776} C_VEL
LIN {X 0,Y 467.345,Z 444.755,A -85,B 0,C 180,E1 -7632.497,E2 -7632.497} C_VEL
LIN {X 0,Y 467.211,Z 451.099,A -85,B 0,C 180,E1 -7634.57,E2 -7634.57} C_VEL
LIN {X 0,Y 469.812,Z 466.696,A -85,B 0,C 180,E1 -7635.088,E2 -7635.088} C_VEL
LIN {X 0,Y 470.137,Z 471.543,A -85,B 0,C 180,E1 -7635.278,E2 -7635.278} C_VEL
LIN {X 0,Y 469.741,Z 483.223,A -85,B 0,C 180,E1 -7635.819,E2 -7635.819} C_VEL
LIN {X 0,Y 469.267,Z 494.459,A -85,B 0,C 180,E1 -7636.5,E2 -7636.5} C_VEL
LIN {X 0,Y 468.852,Z 505.101,A -85,B 0,C 180,E1 -7637.316,E2 -7637.316} C_VEL
LIN {X 0,Y 468.401,Z 515.596,A -85,B 0,C 180,E1 -7638.313,E2 -7638.313} C_VEL
LIN {X 0,Y 467.879,Z 524.785,A -85,B 0,C 180,E1 -7639.397,E2 -7639.397} C_VEL
LIN {X 0,Y 467.447,Z 533.687,A -85,B 0,C 180,E1 -7640.699,E2 -7640.699} C_VEL
LIN {X 0,Y 467.092,Z 540.848,A -85,B 0,C 180,E1 -7642,E2 -7642} C_VEL
LIN {X 0,Y 466.87,Z 547.224,A -85,B 0,C 180,E1 -7643.479,E2 -7643.479} C_VEL
LIN {X 0,Y 466.784,Z 551.676,A -85,B 0,C 180,E1 -7644.817,E2 -7644.817} C_VEL
LIN {X 0,Y 466.663,Z 553.957,A -85,B 0,C 180,E1 -7645.681,E2 -7645.681} C_VEL
LIN {X 0,Y 466.695,Z 555.806,A -85,B 0,C 180,E1 -7646.546,E2 -7646.546} C_VEL
LIN {X 0,Y 466.646,Z 557.192,A -85,B 0,C 180,E1 -7647.41,E2 -7647.41} C_VEL
LIN {X 0,Y 466.589,Z 558.785,A -85,B 0,C 180,E1 -7649.137,E2 -7649.137} C_VEL
LIN {X 0,Y 466.57,Z 559,A -85,B 0,C 180,E1 -7650,E2 -7650} C_VEL
LIN {X 0,Y 466.589,Z 558.786,A -85,B 0,C 180,E1 -7650.863,E2 -7650.863} C_VEL
LIN {X 0,Y 466.646,Z 557.196,A -85,B 0,C 180,E1 -7652.589,E2 -7652.589} C_VEL
LIN {X 0,Y 466.695,Z 555.81,A -85,B 0,C 180,E1 -7653.453,E2 -7653.453} C_VEL
LIN {X 0,Y 466.703,Z 552.896,A -85,B 0,C 180,E1 -7654.751,E2 -7654.751} C_VEL
LIN {X 0,Y 466.839,Z 548.949,A -85,B 0,C 180,E1 -7656.049,E2 -7656.049} C_VEL
LIN {X 0,Y 466.998,Z 542.877,A -85,B 0,C 180,E1 -7657.566,E2 -7657.566} C_VEL
LIN {X 0,Y 467.35,Z 536.237,A -85,B 0,C 180,E1 -7658.866,E2 -7658.866} C_VEL
LIN {X 0,Y 467.739,Z 527.995,A -85,B 0,C 180,E1 -7660.168,E2 -7660.168} C_VEL
LIN {X 0,Y 468.149,Z 519.522,A -85,B 0,C 180,E1 -7661.254,E2 -7661.254} C_VEL
LIN {X 0,Y 468.674,Z 509.158,A -85,B 0,C 180,E1 -7662.323,E2 -7662.323} C_VEL
LIN {X 0,Y 469.089,Z 497.573,A -85,B 0,C 180,E1 -7663.284,E2 -7663.284} C_VEL
LIN {X 0,Y 469.625,Z 485.244,A -85,B 0,C 180,E1 -7664.074,E2 -7664.074} C_VEL
LIN {X 0,Y 470.1,Z 472.877,A -85,B 0,C 180,E1 -7664.667,E2 -7664.667} C_VEL
LIN {X 0,Y 469.979,Z 467.891,A -85,B 0,C 180,E1 -7664.865,E2 -7664.865} C_VEL
LIN {X 0,Y 467.865,Z 455.099,A -85,B 0,C 180,E1 -7665.308,E2 -7665.308} C_VEL
LIN {X 0,Y 467.249,Z 451.178,A -85,B 0,C 180,E1 -7665.428,E2 -7665.428} C_VEL
LIN {X 0,Y 467.484,Z 441.201,A -85,B 0,C 180,E1 -7668.715,E2 -7668.715} C_VEL
LIN {X 0,Y 467.75,Z 431.161,A -85,B 0,C 180,E1 -7672.062,E2 -7672.062} C_VEL
LIN {X 0,Y 468.05,Z 421.682,A -85,B 0,C 180,E1 -7675.298,E2 -7675.298} C_VEL
LIN {X 0,Y 468.402,Z 413.673,A -85,B 0,C 180,E1 -7678.204,E2 -7678.204} C_VEL
LIN {X 0,Y 468.83,Z 404.434,A -85,B 0,C 180,E1 -7681.645,E2 -7681.645} C_VEL
LIN {X 0,Y 469.281,Z 396.581,A -85,B 0,C 180,E1 -7684.686,E2 -7684.686} C_VEL
LIN {X 0,Y 469.422,Z 393.16,A -85,B 0,C 180,E1 -7686.053,E2 -7686.053} C_VEL
LIN {X 0,Y 468.803,Z 388.794,A -85,B 0,C 180,E1 -7687.925,E2 -7687.925} C_VEL
LIN {X 0,Y 467.595,Z 382.242,A -85,B 0,C 180,E1 -7690.971,E2 -7690.971} C_VEL
LIN {X 0,Y 467.55,Z 382.248,A -85,B 0,C 180,E1 -7693.82,E2 -7693.82} C_VEL
LIN {X 0,Y 467.551,Z 382.248,A -85,B 0,C 180,E1 -7696.255,E2 -7696.255} C_VEL
LIN {X 0,Y 467.579,Z 382.244,A -85,B 0,C 180,E1 -7698.721,E2 -7698.721} C_VEL
LIN {X 0,Y 467.571,Z 382.245,A -85,B 0,C 180,E1 -7701.406,E2 -7701.406} C_VEL
LIN {X 0,Y 467.557,Z 382.245,A -85,B 0,C 180,E1 -7704.26,E2 -7704.26} C_VEL
LIN {X 0,Y 467.575,Z 382.244,A -85,B 0,C 180,E1 -7707.32,E2 -7707.32} C_VEL
LIN {X 0,Y 467.563,Z 382.246,A -85,B 0,C 180,E1 -7710.667,E2 -7710.667} C_VEL
LIN {X 0,Y 467.62,Z 382.238,A -85,B 0,C 180,E1 -7713.2,E2 -7713.2} C_VEL
LIN {X 0,Y 467.584,Z 382.243,A -85,B 0,C 180,E1 -7716.468,E2 -7716.468} C_VEL
LIN {X 0,Y 467.615,Z 382.237,A -85,B 0,C 180,E1 -7719.777,E2 -7719.777} C_VEL
LIN {X 0,Y 467.601,Z 382.24,A -85,B 0,C 180,E1 -7722.506,E2 -7722.506} C_VEL
LIN {X 0,Y 467.597,Z 382.24,A -85,B 0,C 180,E1 -7725.196,E2 -7725.196} C_VEL
LIN {X 0,Y 467.647,Z 382.232,A -85,B 0,C 180,E1 -7727.854,E2 -7727.854} C_VEL
